// ---- POUs/VisMain/MAIN_VISION.TcPOU
PROGRAM MAIN_VISION
VAR
	fbPosCam1		: FB_PosImgSts;
	fbPosCam2		: FB_PosImgSts;
	fbPosCam3		: FB_PosImgSts;
	fbPosCam4		: FB_PosImgSts;
	fbPosCam5		: FB_PosImgSts;
	fbPosCam6		: FB_PosImgSts;
	fbPosCam7		: FB_PosImgSts;
	fbPosCam8		: FB_PosImgSts;
	fbPosCam9		: FB_PosImgSts;
	fbPosCam10		: FB_PosImgSts;
	
	fbMidStationCam	: FB_MidStaion;
	fbInfeedCam		: FB_InfeedCam;
	fbOutfeedCam	: FB_OutfeedCam;
	fbRejectCam		: FB_RejectCam;
	stPalletPosData	: ST_PalletImagingData;
	
	stMirrorDataSts1	: ST_Vis_Mirror;
	stMirrorDataSts2	: ST_Vis_Mirror;
	stMirrorDataSts3	: ST_Vis_Mirror;
	stMirrorDataSts4	: ST_Vis_Mirror;
	stMirrorDataSts5	: ST_Vis_Mirror;
	stMirrorDataSts6	: ST_Vis_Mirror;
	stMirrorDataSts7	: ST_Vis_Mirror;
	stMirrorDataSts8	: ST_Vis_Mirror;
	stMirrorDataSts9	: ST_Vis_Mirror;
	stMirrorDataSts10	: ST_Vis_Mirror;
	
	Cam1Trig : R_Trig;
	Cam2Trig : R_Trig;
	Cam3Trig : R_Trig;
	Cam4Trig : R_Trig; 
	Cam5Trig : R_Trig;
	Cam6Trig : R_Trig;
	Cam7Trig : R_Trig; 
	Cam8Trig : R_Trig;
	Cam9Trig : R_Trig; 
	Cam10Trig : R_Trig;
	CamMidStationTrig : R_Trig;
	CamInfeedTrig : R_Trig;
	CamOutfeedTrig : R_Trig;
	CamRejectTrig : R_Trig; 

	ImagingQueStep	: INT;
	
END_VAR


fbPosCam1(iStationId := 1 ,stPosData := stMirrorDataSts1, stAssemblyType := MAIN.stAssemblyData, nX := 830, nY := 980,stModuleHmi := MAIN.stModuleHmi );
fbPosCam2(iStationId := 2 ,stPosData := stMirrorDataSts2, stAssemblyType := MAIN.stAssemblyData, nX := 800, nY := 950,stModuleHmi := MAIN.stModuleHmi  );
fbPosCam3(iStationId := 3 ,stPosData := stMirrorDataSts3, stAssemblyType := MAIN.stAssemblyData, nX := 900, nY := 1010,stModuleHmi := MAIN.stModuleHmi  );
fbPosCam4(iStationId := 4 ,stPosData := stMirrorDataSts4, stAssemblyType := MAIN.stAssemblyData, nX := 890, nY := 950,stModuleHmi := MAIN.stModuleHmi  );
fbPosCam5(iStationId := 5 ,stPosData := stMirrorDataSts5, stAssemblyType := MAIN.stAssemblyData, nX := 840, nY := 1000,stModuleHmi := MAIN.stModuleHmi  );
fbPosCam6(iStationId := 6 ,stPosData := stMirrorDataSts6, stAssemblyType := MAIN.stAssemblyData, nX := 805, nY := 995,stModuleHmi := MAIN.stModuleHmi  );
fbPosCam7(iStationId := 7 ,stPosData := stMirrorDataSts7, stAssemblyType := MAIN.stAssemblyData, nX := 880, nY := 990,stModuleHmi := MAIN.stModuleHmi  );
fbPosCam8(iStationId := 8 ,stPosData := stMirrorDataSts8, stAssemblyType := MAIN.stAssemblyData, nX := 840, nY := 1010,stModuleHmi := MAIN.stModuleHmi  );
fbPosCam9(iStationId := 9 ,stPosData := stMirrorDataSts9, stAssemblyType := MAIN.stAssemblyData, nX := 850, nY := 990,stModuleHmi := MAIN.stModuleHmi  );
fbPosCam10(iStationId := 10 ,stPosData := stMirrorDataSts10, stAssemblyType := MAIN.stAssemblyData, nX := 860, nY := 1000,stModuleHmi := MAIN.stModuleHmi  );

fbMidStationCam(stRecipeData := MAIN.stAssemblyData, iStationId := MAIN.fbMeca500.iWorkingStation, stCouplerData := MAIN.stCouplerData);
fbInfeedCam(stPosData := stPalletPosData, stImagingSetValues := MAIN.stAssemblyData);
fbOutfeedCam();
fbRejectCam();

CASE ImagingQueStep OF
	0: ImagingQueStep := 1;// OFFLINE
	1: CamMidStationTrig(CLK := Trig.bMidStationCam);
		IF CamMidStationTrig.Q THEN
			fbMidStationCam.TrigImage();
		END_IF
		IF NOT Trig.bMidStationCam THEN
			ImagingQueStep := 2;
		END_IF
	2: CamInfeedTrig(CLK := Trig.bInfeedCam);
		IF CamInfeedTrig.Q THEN
			fbInfeedCam.TrigImage();
		END_IF
		IF NOT Trig.bInfeedCam THEN
			ImagingQueStep := 3;
		END_IF
	
	3:	CamOutfeedTrig(CLK := Trig.bOutfeedCam);
		IF CamOutfeedTrig.Q THEN
			fbOutfeedCam.TrigImage();
		END_IF
		IF NOT Trig.bOutfeedCam THEN
			ImagingQueStep := 4;
		END_IF
	
	4:	CamRejectTrig(CLK := Trig.bRejectCam);
		IF CamRejectTrig.Q THEN
			fbRejectCam.TrigImage();
		END_IF
		IF NOT Trig.bRejectCam THEN
			ImagingQueStep := 5;
		END_IF
	5: Cam1Trig(CLK := MAIN.stStation.fbSts1.bTrigPosCam);
		 IF Cam1Trig.Q THEN
			IF MAIN.stStation.fbSts1.bTrigPosCamLightTest THEN
				fbPosCam1.bTrigLightTestImage := TRUE;
			ELSIF MAIN.stStation.fbSts1.bTrigPosCamLaserTest THEN
				fbPosCam1.bTrigLaserTestImage := TRUE;
			ELSIF MAIN.stStation.fbSts1.bTrigPosCamCoupler THEN
				fbPosCam1.bTrigCouplerImage := TRUE;
			END_IF
			fbPosCam1.TrigImage();
		END_IF
		IF NOT MAIN.stStation.fbSts1.bTrigPosCam THEN
			stMirrorDataSts1.bDetectionFailed := FALSE;
			stMirrorDataSts1.bImagingDone := FALSE;
			ImagingQueStep := 6; 
		END_IF
		IF Cam1Trig.CLK THEN
			stMirrorDataSts1.bReadyForTrigger := FALSE;
		ELSE
			stMirrorDataSts1.bReadyForTrigger := TRUE;
		END_IF
		
	6:  Cam2Trig(CLK := MAIN.stStation.fbSts2.bTrigPosCam);
		IF Cam2Trig.Q THEN
			IF MAIN.stStation.fbSts2.bTrigPosCamLightTest THEN
				fbPosCam2.bTrigLightTestImage := TRUE;
			ELSIF MAIN.stStation.fbSts2.bTrigPosCamLaserTest THEN
				fbPosCam2.bTrigLaserTestImage := TRUE;
			ELSIF MAIN.stStation.fbSts2.bTrigPosCamCoupler THEN
				fbPosCam2.bTrigCouplerImage := TRUE;
			END_IF
			fbPosCam2.TrigImage();
		END_IF
	
		IF NOT MAIN.stStation.fbSts2.bTrigPosCam THEN
			stMirrorDataSts2.bDetectionFailed := FALSE;
			stMirrorDataSts2.bImagingDone := FALSE;
			ImagingQueStep := 7;
		END_IF
	
		IF Cam2Trig.CLK THEN
			stMirrorDataSts2.bReadyForTrigger := FALSE;
		ELSE
			stMirrorDataSts2.bReadyForTrigger := TRUE;
		END_IF
	
	
	7:  Cam3Trig(CLK := MAIN.stStation.fbSts3.bTrigPosCam);
		IF Cam3Trig.Q THEN
			IF MAIN.stStation.fbSts3.bTrigPosCamLightTest THEN
				fbPosCam3.bTrigLightTestImage := TRUE;
			ELSIF MAIN.stStation.fbSts3.bTrigPosCamLaserTest THEN
				fbPosCam3.bTrigLaserTestImage := TRUE;
			ELSIF MAIN.stStation.fbSts3.bTrigPosCamCoupler THEN
				fbPosCam3.bTrigCouplerImage := TRUE;
			END_IF
			fbPosCam3.TrigImage();
		END_IF
	
		IF NOT MAIN.stStation.fbSts3.bTrigPosCam THEN
			stMirrorDataSts3.bDetectionFailed := FALSE;
			stMirrorDataSts3.bImagingDone := FALSE;
			ImagingQueStep := 8;
		END_IF
	
		IF Cam3Trig.CLK THEN
			stMirrorDataSts3.bReadyForTrigger := FALSE;
		ELSE
			stMirrorDataSts3.bReadyForTrigger := TRUE;
		END_IF
	
	
	8:  Cam4Trig(CLK := MAIN.stStation.fbSts4.bTrigPosCam);
		IF Cam4Trig.Q THEN
			IF MAIN.stStation.fbSts4.bTrigPosCamLightTest THEN
				fbPosCam4.bTrigLightTestImage := TRUE;
			ELSIF MAIN.stStation.fbSts4.bTrigPosCamLaserTest THEN
				fbPosCam4.bTrigLaserTestImage := TRUE;
			ELSIF MAIN.stStation.fbSts4.bTrigPosCamCoupler THEN
				fbPosCam4.bTrigCouplerImage := TRUE;
			END_IF
			fbPosCam4.TrigImage();
		END_IF
	
		IF NOT MAIN.stStation.fbSts4.bTrigPosCam THEN
			stMirrorDataSts4.bDetectionFailed := FALSE;
			stMirrorDataSts4.bImagingDone := FALSE;
			ImagingQueStep := 9;
		END_IF
	
		IF Cam4Trig.CLK THEN
			stMirrorDataSts4.bReadyForTrigger := FALSE;
		ELSE
			stMirrorDataSts4.bReadyForTrigger := TRUE;
		END_IF
	
	
	9:  Cam5Trig(CLK := MAIN.stStation.fbSts5.bTrigPosCam);
		IF Cam5Trig.Q THEN
			IF MAIN.stStation.fbSts5.bTrigPosCamLightTest THEN
				fbPosCam5.bTrigLightTestImage := TRUE;
			ELSIF MAIN.stStation.fbSts5.bTrigPosCamLaserTest THEN
				fbPosCam5.bTrigLaserTestImage := TRUE;
			ELSIF MAIN.stStation.fbSts5.bTrigPosCamCoupler THEN
				fbPosCam5.bTrigCouplerImage := TRUE;
			END_IF
			fbPosCam5.TrigImage();
		END_IF
	
		IF NOT MAIN.stStation.fbSts5.bTrigPosCam THEN
			stMirrorDataSts5.bDetectionFailed := FALSE;
			stMirrorDataSts5.bImagingDone := FALSE;
			ImagingQueStep := 10;
		END_IF
	
		IF Cam5Trig.CLK THEN
			stMirrorDataSts5.bReadyForTrigger := FALSE;
		ELSE
			stMirrorDataSts5.bReadyForTrigger := TRUE;
		END_IF
	
	
	10: Cam6Trig(CLK := MAIN.stStation.fbSts6.bTrigPosCam);
		IF Cam6Trig.Q THEN
			IF MAIN.stStation.fbSts6.bTrigPosCamLightTest THEN
				fbPosCam6.bTrigLightTestImage := TRUE;
			ELSIF MAIN.stStation.fbSts6.bTrigPosCamLaserTest THEN
				fbPosCam6.bTrigLaserTestImage := TRUE;
			ELSIF MAIN.stStation.fbSts6.bTrigPosCamCoupler THEN
				fbPosCam6.bTrigCouplerImage := TRUE;
			END_IF
			fbPosCam6.TrigImage();
		END_IF
	
		IF NOT MAIN.stStation.fbSts6.bTrigPosCam THEN
			stMirrorDataSts6.bDetectionFailed := FALSE;
			stMirrorDataSts6.bImagingDone := FALSE;
			ImagingQueStep := 11;
		END_IF
	
		IF Cam6Trig.CLK THEN
			stMirrorDataSts6.bReadyForTrigger := FALSE;
		ELSE
			stMirrorDataSts6.bReadyForTrigger := TRUE;
		END_IF
	
	
	11: Cam7Trig(CLK := MAIN.stStation.fbSts7.bTrigPosCam);
		IF Cam7Trig.Q THEN
			IF MAIN.stStation.fbSts7.bTrigPosCamLightTest THEN
				fbPosCam7.bTrigLightTestImage := TRUE;
			ELSIF MAIN.stStation.fbSts7.bTrigPosCamLaserTest THEN
				fbPosCam7.bTrigLaserTestImage := TRUE;
			ELSIF MAIN.stStation.fbSts7.bTrigPosCamCoupler THEN
				fbPosCam7.bTrigCouplerImage := TRUE;
			END_IF
			fbPosCam7.TrigImage();
		END_IF
	
		IF NOT MAIN.stStation.fbSts7.bTrigPosCam THEN
			stMirrorDataSts7.bDetectionFailed := FALSE;
			stMirrorDataSts7.bImagingDone := FALSE;
			ImagingQueStep := 12;
		END_IF
	
		IF Cam7Trig.CLK THEN
			stMirrorDataSts7.bReadyForTrigger := FALSE;
		ELSE
			stMirrorDataSts7.bReadyForTrigger := TRUE;
		END_IF
	
	
	12: Cam8Trig(CLK := MAIN.stStation.fbSts8.bTrigPosCam);
		IF Cam8Trig.Q THEN
			IF MAIN.stStation.fbSts8.bTrigPosCamLightTest THEN
				fbPosCam8.bTrigLightTestImage := TRUE;
			ELSIF MAIN.stStation.fbSts8.bTrigPosCamLaserTest THEN
				fbPosCam8.bTrigLaserTestImage := TRUE;
			ELSIF MAIN.stStation.fbSts8.bTrigPosCamCoupler THEN
				fbPosCam8.bTrigCouplerImage := TRUE;
			END_IF
			fbPosCam8.TrigImage();
		END_IF
	
		IF NOT MAIN.stStation.fbSts8.bTrigPosCam THEN
			stMirrorDataSts8.bDetectionFailed := FALSE;
			stMirrorDataSts8.bImagingDone := FALSE;
			ImagingQueStep := 13;
		END_IF
	
		IF Cam8Trig.CLK THEN
			stMirrorDataSts8.bReadyForTrigger := FALSE;
		ELSE
			stMirrorDataSts8.bReadyForTrigger := TRUE;
		END_IF
	
	
	13: Cam9Trig(CLK := MAIN.stStation.fbSts9.bTrigPosCam);
		IF Cam9Trig.Q THEN
			IF MAIN.stStation.fbSts9.bTrigPosCamLightTest THEN
				fbPosCam9.bTrigLightTestImage := TRUE;
			ELSIF MAIN.stStation.fbSts9.bTrigPosCamLaserTest THEN
				fbPosCam9.bTrigLaserTestImage := TRUE;
			ELSIF MAIN.stStation.fbSts9.bTrigPosCamCoupler THEN
				fbPosCam9.bTrigCouplerImage := TRUE;
			END_IF
			fbPosCam9.TrigImage();
		END_IF
	
		IF NOT MAIN.stStation.fbSts9.bTrigPosCam THEN
			stMirrorDataSts9.bDetectionFailed := FALSE;
			stMirrorDataSts9.bImagingDone := FALSE;
			ImagingQueStep := 14;
		END_IF
	
		IF Cam9Trig.CLK THEN
			stMirrorDataSts9.bReadyForTrigger := FALSE;
		ELSE
			stMirrorDataSts9.bReadyForTrigger := TRUE;
		END_IF
	
	
	14: Cam10Trig(CLK := MAIN.stStation.fbSts10.bTrigPosCam);
		IF Cam10Trig.Q THEN
			IF MAIN.stStation.fbSts10.bTrigPosCamLightTest THEN
				fbPosCam10.bTrigLightTestImage := TRUE;
			ELSIF MAIN.stStation.fbSts10.bTrigPosCamLaserTest THEN
				fbPosCam10.bTrigLaserTestImage := TRUE;
			ELSIF MAIN.stStation.fbSts10.bTrigPosCamCoupler THEN
				fbPosCam10.bTrigCouplerImage := TRUE;
			END_IF
			fbPosCam10.TrigImage();
		END_IF
	
		IF NOT MAIN.stStation.fbSts10.bTrigPosCam THEN
			stMirrorDataSts10.bDetectionFailed := FALSE;
			stMirrorDataSts10.bImagingDone := FALSE;
			ImagingQueStep := 15;
		END_IF
	
		IF Cam10Trig.CLK THEN
			stMirrorDataSts10.bReadyForTrigger := FALSE;
		ELSE
			stMirrorDataSts10.bReadyForTrigger := TRUE;
		END_IF

	15: ImagingQueStep := 1;
	22: IF Trig.bInfeedCam THEN
			fbInfeedCam.TrigImage();
			Trig.bInfeedCam := FALSE;
		END_IF
END_CASE

END_PROGRAM

// ---- POUs/Sts/Vis/FB_PosImgSts.TcPOU
FUNCTION_BLOCK FB_PosImgSts
VAR_INPUT
	bTrigLightTestImage	: BOOL;
	bTrigLaserTestImage	: BOOL;
	bTrigCouplerImage		: BOOL;
	stPosData	: REFERENCE TO ST_Vis_Mirror;
	stAssemblyType : REFERENCE TO ST_Recipes;
	nX		: UDINT;
	nY		: UDINT;
	iStationId	: INT;
	stModuleHmi	: REFERENCE TO ST_ModuleHmi;
END_VAR
VAR_OUTPUT
	bImageReceived : BOOL;
	bPartDetectFailed : BOOL;
	iErrorId			: INT;
	bDone : BOOL;
END_VAR
VAR
	hr									: HRESULT;
	eVisionState						: ETcVnCameraState;
	fbCamera          					: FB_VN_GevCameraControl;
	ImageRawDisp						: ITcVnDisplayableImage;
	nNewImageCounter 					: UINT;
	ImageRaw							: Tc3_Vision.ITcVnImage;
	ipImageProsessed					: Tc3_Vision.ITcVnImage;
	ipImageProsessedDisp				: Tc3_Vision.ITcVnDisplayableImage;
	ipImageTest							: ITcVnImage;
	ipImageTestDisp						: ITcVnDisplayableImage;

	aStartPointCoupler1 				: TcVnPoint2_REAL;
	aEndPointCoupler1					: TcVnPoint2_REAL;
	
	ipEdgePointsCoupler1   				: ITcVnContainer;
	ipEdgePointsCoupler2				: ITcVnContainer;
	ipEdgePointsCoupler3				: ITcVnContainer;
	
	aStartPointCoupler2 				: TcVnPoint2_REAL;
	aEndPointCoupler2					: TcVnPoint2_REAL;
	aStartPointCoupler3 				: TcVnPoint2_REAL;
	aEndPointCoupler3					: TcVnPoint2_REAL;
	
	aStartPointMirror1 					: TcVnPoint2_REAL;
	aEndPointMirror1					: TcVnPoint2_REAL;
	aStartPointMirror2 					: TcVnPoint2_REAL;
	aEndPointMirror2					: TcVnPoint2_REAL;
	ipEdgePointsMirror1   				: ITcVnContainer;
	ipEdgePointsMirror2   				: ITcVnContainer;
	aElementMirror1						: TcVnPoint2_REAL;
	aElementMirror2						: TcVnPoint2_REAL;
	
	aMirrorEdgeCalc			: TcVnPoint2_REAL;
	aMirrorEdgeReal			: TcVnPoint2_REAL;
	

	
	rThreshold			: LREAL := 45;
	rMaxvalue			: LREAL := 255;

	stDetectionAreaLed						: TcVnRectangle_UDINT;
	stDetectionAreaLaser					: TcVnRectangle_UDINT;
	aAverageLed  							: TcVnVector4_LREAL;
	aAverageLaser  							: TcVnVector4_LREAL;
	aElementCoupler1 						: TcVnPoint2_REAL; 
	aElementCoupler2						: ARRAY [0..5] OF TcVnPoint2_REAL;
	aElementCoupler3						: ARRAY [0..5] OF TcVnPoint2_REAL;
	aCouplerAverage2						: TcVnPoint2_REAL;
	aCouplerAverage3						: TcVnPoint2_REAL;
	aCouplerCenterpoint						: TcVnPoint2_REAL;
	rWorldDistance							: LREAL;
	fbEventlogger							: FB_EventLogger;
	bInitTrig 								: BOOL;
	TrigCheckTmr							: TON;
END_VAR

fbEventlogger(stModuleHmi:=stModuleHmi);
eVisionState := fbCamera.GetState();

stDetectionAreaLed.nHeight := 200;
stDetectionAreaLed.nWidth := 200;
stDetectionAreaLed.nX := 1800;
stDetectionAreaLed.nY := 900;

stDetectionAreaLaser.nHeight := 20;
stDetectionAreaLaser.nWidth := 20;
stDetectionAreaLaser.nX := nX;
stDetectionAreaLaser.nY := nY;

bDone := FALSE;
bImageReceived := FALSE;
hr := 0;
TrigCheckTmr(PT := T#1S);


IF eVisionState = TCVN_CS_ERROR THEN
	hr := fbCamera.Reset();
ELSIF eVisionState = TCVN_CS_TRIGGERING THEN
	hr := fbCamera.TriggerImage();
ELSIF eVisionState < TCVN_CS_ACQUIRING THEN
    hr := fbCamera.StartAcquisition();
ELSIF eVisionState = TCVN_CS_ACQUIRING THEN
	hr := fbCamera.GetCurrentImageUndistorted(ImageRaw); 
	IF SUCCEEDED(hr) AND ImageRaw <> 0 THEN
		bPartDetectFailed := FALSE;
		bImageReceived := TRUE;
		nNewImageCounter := nNewImageCounter +1;
// 		hr := F_VN_CopyImage(ImageRaw, ipImageProsessed, hr);
// 		hr := F_VN_CopyIntoDisplayableImage (ImageRaw, ImageRawDisp, hr);
		bInitTrig := FALSE;
		TrigCheckTmr.IN := FALSE;
		hr := F_VN_ConvertColorSpace(ipSrcImage:= ImageRaw , ipDestImage:= ipImageProsessed ,
			eTransform:= ETcVnColorSpaceTransform.TCVN_CST_GRAY_TO_RGB, hrPrev:= hr);
		IF bTrigLightTestImage THEN
			hr := F_VN_CopyImage(ImageRaw, ipImageTest, hrPrev := hr);
			hr := F_VN_SetRoi_TcVnRectangle_UDINT(stRoi:= stDetectionAreaLed, ipDestImage:= ipImageTest, hrPrev:= hr);
			hr := F_VN_ImageAverage(ipSrcImage:= ipImageTest, aAverage:= aAverageLed, hrPrev:= hr);
			hr := F_VN_ResetRoi(ipImage:= ipImageTest, hrPrev:= hr);
			hr:= F_VN_ConvertColorSpace(ipSrcImage:= ipImageTest , ipDestImage:= ipImageTest ,
				eTransform:= ETcVnColorSpaceTransform.TCVN_CST_GRAY_TO_RGB, hrPrev:= hr);
			hr := F_VN_DrawRectangle_TcVnRectangle_UDINT(
				stRectangle:= stDetectionAreaLed,
				ipDestImage:= ipImageTest,
				aColor:= Color.Green,
				nThickness:= 1,
				hrPrev:= hr);
			hr := F_VN_CopyIntoDisplayableImage (ipImageTest, ipImageTestDisp, hr);	
			IF aAverageLed[0] > 230 THEN
				stPosData.bLightTestOk := TRUE;
				stPosData.bDetectionFailed := FALSE;
			ELSE
				stPosData.bLightTestOk := FALSE;
				stPosData.bDetectionFailed := TRUE;
			END_IF
			bTrigLightTestImage := FALSE;
		ELSIF bTrigLaserTestImage THEN
			hr := F_VN_CopyImage(ImageRaw, ipImageTest, hrPrev := hr);
			hr := F_VN_SetRoi_TcVnRectangle_UDINT(stRoi:= stDetectionAreaLaser, ipDestImage:= ipImageTest, hrPrev:= hr);
			hr := F_VN_ImageAverage(ipSrcImage:= ipImageTest, aAverage:= aAverageLaser, hrPrev:= hr);
			hr := F_VN_ResetRoi(ipImage:= ipImageTest, hrPrev:= hr);
			hr:= F_VN_ConvertColorSpace(ipSrcImage:= ipImageTest , ipDestImage:= ipImageTest ,
				eTransform:= ETcVnColorSpaceTransform.TCVN_CST_GRAY_TO_RGB, hrPrev:= hr);
			hr := F_VN_DrawRectangle_TcVnRectangle_UDINT(
				stRectangle:= stDetectionAreaLaser,
				ipDestImage:= ipImageTest,
				aColor:= Color.Green,
				nThickness:= 1,
				hrPrev:= hr);
			hr := F_VN_CopyIntoDisplayableImage (ipImageTest, ipImageTestDisp, hr);	
			IF aAverageLaser[0] > 230 THEN
				stPosData.bLaserTestOk := TRUE;
				stPosData.bDetectionFailed := FALSE;
			ELSE
				stPosData.bLaserTestOk := FALSE;
				stPosData.bDetectionFailed := TRUE;
			END_IF
			bTrigLaserTestImage := FALSE;
		ELSIF bTrigCouplerImage THEN	
			CouplerDetect();			
			bTrigCouplerImage := FALSE;
			stPosData.bImagingDone := TRUE;		
		ELSE
 			MirrorDetect();
			stPosData.bImagingDone := TRUE;	
		END_IF
	ELSIF bInitTrig AND TrigCheckTmr.Q THEN
		iErrorId := 304;
		fbEventlogger.bRaiseAlarm[11]:=TRUE;
		fbEventlogger.sErrorCode:= CONCAT(CONCAT('3', INT_TO_STRING(iStationId)), '4');
		bInitTrig := FALSE;
		TrigCheckTmr.IN := FALSE;
	END_IF
END_IF

METHOD CheckType : BOOL
VAR_INPUT
END_VAR
// CASE iStationId OF
// 	1..5: 
// 		IF stAssemblyType.Station1To5.sAssemblyType = 'AL-86068' THEN
// 			aStartPointCoupler1[0] := 750;
// 			aStartPointCoupler1[1] := 800;
// 			aEndPointCoupler1[0] := 750;
// 			aEndPointCoupler1[1] := 900;
// 			
// 			aStartPointCoupler2[0] := 750;
// 			aStartPointCoupler2[1] := 1170;
// 			aEndPointCoupler2[0] := 750;
// 			aEndPointCoupler2[1] := 1090;
// 		
// 			aStartPointMirror1[0] := 0;
// 			aStartPointMirror1[1] := 0;
// 			aEndPointMirror1[0] := 0;
// 			aEndPointMirror1[1] := 0;
// 			
// 			aStartPointMirror2[0] := 0;
// 			aStartPointMirror2[1] := 0;
// 			aEndPointMirror2[0] := 0;
// 			aEndPointMirror2[1] := 0;
// 		
// 		ELSIF stAssemblyType.Station1To5.sAssemblyType = 'AL-79710' THEN
// 			aStartPointCoupler1[0] := 770;
// 			aStartPointCoupler1[1] := 840;
// 			aEndPointCoupler1[0] := 770;
// 			aEndPointCoupler1[1] := 920;
// 			
// 			aStartPointCoupler2[0] := 770;
// 			aStartPointCoupler2[1] := 1150;
// 			aEndPointCoupler2[0] := 770;
// 			aEndPointCoupler2[1] := 1050;
// 		
// 			aStartPointMirror1[0] := 0;
// 			aStartPointMirror1[1] := 0;
// 			aEndPointMirror1[0] := 0;
// 			aEndPointMirror1[1] := 0;
// 			
// 			aStartPointMirror2[0] := 0;
// 			aStartPointMirror2[1] := 0;
// 			aEndPointMirror2[0] := 0;
// 			aEndPointMirror2[1] := 0;
// 		
// 		ELSIF stAssemblyType.Station1To5.sAssemblyType = 'AL-82028' THEN
// 			
// 			aStartPointCoupler1[0] := 750;
// 			aStartPointCoupler1[1] := 800;
// 			aEndPointCoupler1[0] := 750;
// 			aEndPointCoupler1[1] := 900;
// 			
// 			aStartPointCoupler2[0] := 750;
// 			aStartPointCoupler2[1] := 1170;
// 			aEndPointCoupler2[0] := 750;
// 			aEndPointCoupler2[1] := 1090;
// 		
// 			aStartPointMirror1[0] := 0;
// 			aStartPointMirror1[1] := 0;
// 			aEndPointMirror1[0] := 0;
// 			aEndPointMirror1[1] := 0;
// 			
// 			aStartPointMirror2[0] := 0;
// 			aStartPointMirror2[1] := 0;
// 			aEndPointMirror2[0] := 0;
// 			aEndPointMirror2[1] := 0;
// 		
// 		ELSIF stAssemblyType.Station1To5.sAssemblyType = 'AL-82026' THEN
// 			aStartPointCoupler[0] := ;
// 			aStartPointCoupler[1] := ;
// 			aEndPointCoupler[0] := ;
// 			aEndPointCoupler[1] := ;
// 		
// 			aStartPointMirror[0] := ;
// 			aStartPointMirror[1] := ;
// 			aEndPointMirror[0] := ;
// 			aEndPointMirror[1] := ;
// 		
// 		ELSIF stAssemblyType.Station1To5.sAssemblyType = 'AL-69219' THEN
// 			aStartPointCoupler1[0] := 793;
// 			aStartPointCoupler1[1] := 680;
// 			aEndPointCoupler1[0] := 793;
// 			aEndPointCoupler1[1] := 780;
// 			
// 			aStartPointCoupler2[0] := 793;
// 			aStartPointCoupler2[1] := 1330;
// 			aEndPointCoupler2[0] := 793;
// 			aEndPointCoupler2[1] := 1200;
// 		
// 			aStartPointMirror1[0] := 0;
// 			aStartPointMirror1[1] := 0;
// 			aEndPointMirror1[0] := 0;
// 			aEndPointMirror1[1] := 0;
// 			
// 			aStartPointMirror2[0] := 0;
// 			aStartPointMirror2[1] := 0;
// 			aEndPointMirror2[0] := 0;
// 			aEndPointMirror2[1] := 0;
// 		
// 		ELSIF stAssemblyType.Station1To5.sAssemblyType = 'AL-71449' THEN
// 			aStartPointCoupler[0] := ;
// 			aStartPointCoupler[1] := ;
// 			aEndPointCoupler[0] := ;
// 			aEndPointCoupler[1] := ;
// 		
// 			aStartPointMirror[0] := ;
// 			aStartPointMirror[1] := ;
// 			aEndPointMirror[0] := ;
// 			aEndPointMirror[1] := ;
// 		
// 		ELSIF stAssemblyType.Station1To5.sAssemblyType = 'AL-70918' THEN
// 			aStartPointCoupler[0] := ;
// 			aStartPointCoupler[1] := ;
// 			aEndPointCoupler[0] := ;
// 			aEndPointCoupler[1] := ;
// 		
// 			aStartPointMirror[0] := ;
// 			aStartPointMirror[1] := ;
// 			aEndPointMirror[0] := ;
// 			aEndPointMirror[1] := ;
// 		
// 		ELSIF stAssemblyType.Station1To5.sAssemblyType = 'AL-200617' THEN
// 			aStartPointCoupler1[0] := 770;
// 			aStartPointCoupler1[1] := 840;
// 			aEndPointCoupler1[0] := 770;
// 			aEndPointCoupler1[1] := 920;
// 			
// 			aStartPointCoupler2[0] := 770;
// 			aStartPointCoupler2[1] := 1150;
// 			aEndPointCoupler2[0] := 770;
// 			aEndPointCoupler2[1] := 1050;
// 		
// 			aStartPointMirror1[0] := 0;
// 			aStartPointMirror1[1] := 0;
// 			aEndPointMirror1[0] := 0;
// 			aEndPointMirror1[1] := 0;
// 			
// 			aStartPointMirror2[0] := 0;
// 			aStartPointMirror2[1] := 0;
// 			aEndPointMirror2[0] := 0;
// 			aEndPointMirror2[1] := 0;
// 		
// 		ELSIF stAssemblyType.Station1To5.sAssemblyType = 'AL-200613' THEN
// 			aStartPointCoupler1[0] := 793;
// 			aStartPointCoupler1[1] := 680;
// 			aEndPointCoupler1[0] := 793;
// 			aEndPointCoupler1[1] := 780;
// 			
// 			aStartPointCoupler2[0] := 793;
// 			aStartPointCoupler2[1] := 1330;
// 			aEndPointCoupler2[0] := 793;
// 			aEndPointCoupler2[1] := 1200;
// 		
// 			aStartPointMirror1[0] := 0;
// 			aStartPointMirror1[1] := 0;
// 			aEndPointMirror1[0] := 0;
// 			aEndPointMirror1[1] := 0;
// 			
// 			aStartPointMirror2[0] := 0;
// 			aStartPointMirror2[1] := 0;
// 			aEndPointMirror2[0] := 0;
// 			aEndPointMirror2[1] := 0;
// 		
// 		ELSIF stAssemblyType.Station1To5.sAssemblyType = 'AL-88450' THEN
// 			aStartPointCoupler[0] := ;
// 			aStartPointCoupler[1] := ;
// 			aEndPointCoupler[0] := ;
// 			aEndPointCoupler[1] := ;
// 		
// 			aStartPointMirror[0] := ;
// 			aStartPointMirror[1] := ;
// 			aEndPointMirror[0] := ;
// 			aEndPointMirror[1] := ;
// 		
// 		ELSIF stAssemblyType.Station1To5.sAssemblyType = 'AL-200665' THEN
// 			aStartPointCoupler1[0] := 644;
// 			aStartPointCoupler1[1] := 780;
// 			aEndPointCoupler1[0] := 644;
// 			aEndPointCoupler1[1] := 780;
// 			
// 			aStartPointCoupler2[0] := 644;
// 			aStartPointCoupler2[1] := 1210;
// 			aEndPointCoupler2[0] := 644;
// 			aEndPointCoupler2[1] := 1100;
// 		
// 			aStartPointMirror1[0] := 0;
// 			aStartPointMirror1[1] := 0;
// 			aEndPointMirror1[0] := 0;
// 			aEndPointMirror1[1] := 0;
// 			
// 			aStartPointMirror2[0] := 0;
// 			aStartPointMirror2[1] := 0;
// 			aEndPointMirror2[0] := 0;
// 			aEndPointMirror2[1] := 0;
// 		
// 		ELSIF stAssemblyType.Station1To5.sAssemblyType = 'AL-200663' THEN
// 			aStartPointCoupler1[0] := 644;
// 			aStartPointCoupler1[1] := 780;
// 			aEndPointCoupler1[0] := 644;
// 			aEndPointCoupler1[1] := 780;
// 			
// 			aStartPointCoupler2[0] := 644;
// 			aStartPointCoupler2[1] := 1210;
// 			aEndPointCoupler2[0] := 644;
// 			aEndPointCoupler2[1] := 1100;
// 		
// 			aStartPointMirror1[0] := 0;
// 			aStartPointMirror1[1] := 0;
// 			aEndPointMirror1[0] := 0;
// 			aEndPointMirror1[1] := 0;
// 			
// 			aStartPointMirror2[0] := 0;
// 			aStartPointMirror2[1] := 0;
// 			aEndPointMirror2[0] := 0;
// 			aEndPointMirror2[1] := 0;
// 		
// 		ELSIF stAssemblyType.Station1To5.sAssemblyType = 'AL-82029' THEN
// 			aStartPointCoupler1[0] := 750;
// 			aStartPointCoupler1[1] := 800;
// 			aEndPointCoupler1[0] := 750;
// 			aEndPointCoupler1[1] := 900;
// 			
// 			aStartPointCoupler2[0] := 750;
// 			aStartPointCoupler2[1] := 1170;
// 			aEndPointCoupler2[0] := 750;
// 			aEndPointCoupler2[1] := 1090;
// 		
// 			aStartPointMirror1[0] := 0;
// 			aStartPointMirror1[1] := 0;
// 			aEndPointMirror1[0] := 0;
// 			aEndPointMirror1[1] := 0;
// 			
// 			aStartPointMirror2[0] := 0;
// 			aStartPointMirror2[1] := 0;
// 			aEndPointMirror2[0] := 0;
// 			aEndPointMirror2[1] := 0;
// 		
// 		ELSIF stAssemblyType.Station1To5.sAssemblyType = 'AL-86069' THEN
// 			aStartPointCoupler1[0] := 750;
// 			aStartPointCoupler1[1] := 800;
// 			aEndPointCoupler1[0] := 750;
// 			aEndPointCoupler1[1] := 900;
// 			
// 			aStartPointCoupler2[0] := 750;
// 			aStartPointCoupler2[1] := 1170;
// 			aEndPointCoupler2[0] := 750;
// 			aEndPointCoupler2[1] := 1090;
// 		
// 			aStartPointMirror1[0] := 0;
// 			aStartPointMirror1[1] := 0;
// 			aEndPointMirror1[0] := 0;
// 			aEndPointMirror1[1] := 0;
// 			
// 			aStartPointMirror2[0] := 0;
// 			aStartPointMirror2[1] := 0;
// 			aEndPointMirror2[0] := 0;
// 			aEndPointMirror2[1] := 0;
// 		
// 		ELSIF stAssemblyType.Station1To5.sAssemblyType = 'AL-79420' THEN
// 			aStartPointCoupler1[0] := 770;
// 			aStartPointCoupler1[1] := 840;
// 			aEndPointCoupler1[0] := 770;
// 			aEndPointCoupler1[1] := 920;
// 			
// 			aStartPointCoupler2[0] := 770;
// 			aStartPointCoupler2[1] := 1150;
// 			aEndPointCoupler2[0] := 770;
// 			aEndPointCoupler2[1] := 1050;
// 		
// 			aStartPointMirror1[0] := 0;
// 			aStartPointMirror1[1] := 0;
// 			aEndPointMirror1[0] := 0;
// 			aEndPointMirror1[1] := 0;
// 			
// 			aStartPointMirror2[0] := 0;
// 			aStartPointMirror2[1] := 0;
// 			aEndPointMirror2[0] := 0;
// 			aEndPointMirror2[1] := 0;
// 		
// 		ELSIF stAssemblyType.Station1To5.sAssemblyType = 'AL-82027' THEN
// 			aStartPointCoupler[0] := ;
// 			aStartPointCoupler[1] := ;
// 			aEndPointCoupler[0] := ;
// 			aEndPointCoupler[1] := ;
// 		
// 			aStartPointMirror[0] := ;
// 			aStartPointMirror[1] := ;
// 			aEndPointMirror[0] := ;
// 			aEndPointMirror[1] := ;
// 		
// 		ELSIF stAssemblyType.Station1To5.sAssemblyType = 'AL-69220' THEN
// 			aStartPointCoupler1[0] := 793;
// 			aStartPointCoupler1[1] := 680;
// 			aEndPointCoupler1[0] := 793;
// 			aEndPointCoupler1[1] := 780;
// 			
// 			aStartPointCoupler2[0] := 793;
// 			aStartPointCoupler2[1] := 1330;
// 			aEndPointCoupler2[0] := 793;
// 			aEndPointCoupler2[1] := 1200;
// 		
// 			aStartPointMirror1[0] := 0;
// 			aStartPointMirror1[1] := 0;
// 			aEndPointMirror1[0] := 0;
// 			aEndPointMirror1[1] := 0;
// 			
// 			aStartPointMirror2[0] := 0;
// 			aStartPointMirror2[1] := 0;
// 			aEndPointMirror2[0] := 0;
// 			aEndPointMirror2[1] := 0;
// 		
// 		ELSIF stAssemblyType.Station1To5.sAssemblyType = 'AL-71450' THEN
// 			aStartPointCoupler[0] := ;
// 			aStartPointCoupler[1] := ;
// 			aEndPointCoupler[0] := ;
// 			aEndPointCoupler[1] := ;
// 		
// 			aStartPointMirror[0] := ;
// 			aStartPointMirror[1] := ;
// 			aEndPointMirror[0] := ;
// 			aEndPointMirror[1] := ;
// 		
// 		ELSIF stAssemblyType.Station1To5.sAssemblyType = 'AL-70916' THEN
// 			aStartPointCoupler[0] := ;
// 			aStartPointCoupler[1] := ;
// 			aEndPointCoupler[0] := ;
// 			aEndPointCoupler[1] := ;
// 		
// 			aStartPointMirror[0] := ;
// 			aStartPointMirror[1] := ;
// 			aEndPointMirror[0] := ;
// 			aEndPointMirror[1] := ;
// 		
// 		ELSIF stAssemblyType.Station1To5.sAssemblyType = 'AL-200618' THEN
// 			aStartPointCoupler1[0] := 770;
// 			aStartPointCoupler1[1] := 840;
// 			aEndPointCoupler1[0] := 770;
// 			aEndPointCoupler1[1] := 920;
// 			
// 			aStartPointCoupler2[0] := 770;
// 			aStartPointCoupler2[1] := 1150;
// 			aEndPointCoupler2[0] := 770;
// 			aEndPointCoupler2[1] := 1050;
// 		
// 			aStartPointMirror1[0] := 0;
// 			aStartPointMirror1[1] := 0;
// 			aEndPointMirror1[0] := 0;
// 			aEndPointMirror1[1] := 0;
// 			
// 			aStartPointMirror2[0] := 0;
// 			aStartPointMirror2[1] := 0;
// 			aEndPointMirror2[0] := 0;
// 			aEndPointMirror2[1] := 0;
// 		
// 		ELSIF stAssemblyType.Station1To5.sAssemblyType = 'AL-200614' THEN
// 			aStartPointCoupler1[0] := 793;
// 			aStartPointCoupler1[1] := 680;
// 			aEndPointCoupler1[0] := 793;
// 			aEndPointCoupler1[1] := 780;
// 			
// 			aStartPointCoupler2[0] := 793;
// 			aStartPointCoupler2[1] := 1330;
// 			aEndPointCoupler2[0] := 793;
// 			aEndPointCoupler2[1] := 1200;
// 		
// 			aStartPointMirror1[0] := 0;
// 			aStartPointMirror1[1] := 0;
// 			aEndPointMirror1[0] := 0;
// 			aEndPointMirror1[1] := 0;
// 			
// 			aStartPointMirror2[0] := 0;
// 			aStartPointMirror2[1] := 0;
// 			aEndPointMirror2[0] := 0;
// 			aEndPointMirror2[1] := 0;
// 		
// 		ELSIF stAssemblyType.Station1To5.sAssemblyType = 'AL-88470' THEN
// 			aStartPointCoupler[0] := ;
// 			aStartPointCoupler[1] := ;
// 			aEndPointCoupler[0] := ;
// 			aEndPointCoupler[1] := ;
// 		
// 			aStartPointMirror[0] := ;
// 			aStartPointMirror[1] := ;
// 			aEndPointMirror[0] := ;
// 			aEndPointMirror[1] := ;
// 		
// 		ELSIF stAssemblyType.Station1To5.sAssemblyType = 'AL-200662' THEN
// 			aStartPointCoupler1[0] := 644;
// 			aStartPointCoupler1[1] := 780;
// 			aEndPointCoupler1[0] := 644;
// 			aEndPointCoupler1[1] := 780;
// 			
// 			aStartPointCoupler2[0] := 644;
// 			aStartPointCoupler2[1] := 1210;
// 			aEndPointCoupler2[0] := 644;
// 			aEndPointCoupler2[1] := 1100;
// 		
// 			aStartPointMirror1[0] := 0;
// 			aStartPointMirror1[1] := 0;
// 			aEndPointMirror1[0] := 0;
// 			aEndPointMirror1[1] := 0;
// 			
// 			aStartPointMirror2[0] := 0;
// 			aStartPointMirror2[1] := 0;
// 			aEndPointMirror2[0] := 0;
// 			aEndPointMirror2[1] := 0;
// 		
// 		ELSIF stAssemblyType.Station1To5.sAssemblyType = 'AL-200664' THEN
// 			aStartPointCoupler1[0] := 644;
// 			aStartPointCoupler1[1] := 780;
// 			aEndPointCoupler1[0] := 644;
// 			aEndPointCoupler1[1] := 780;
// 			
// 			aStartPointCoupler2[0] := 644;
// 			aStartPointCoupler2[1] := 1210;
// 			aEndPointCoupler2[0] := 644;
// 			aEndPointCoupler2[1] := 1100;
// 		
// 			aStartPointMirror1[0] := 0;
// 			aStartPointMirror1[1] := 0;
// 			aEndPointMirror1[0] := 0;
// 			aEndPointMirror1[1] := 0;
// 			
// 			aStartPointMirror2[0] := 0;
// 			aStartPointMirror2[1] := 0;
// 			aEndPointMirror2[0] := 0;
// 			aEndPointMirror2[1] := 0;
// 		
// 		END_IF;
// 
// END_CASE
END_METHOD

METHOD CouplerDetect : BOOL

VAR
	bCheckOnce 					: BOOL := TRUE;
	hrEdgeT						: HRESULT;
	nIndex						: ULINT;
	
END_VAR
hrEdgeT := 0;

aStartPointCoupler1[0] := 1000;
aStartPointCoupler1[1] := 1000;
aEndPointCoupler1[0] := 550;
aEndPointCoupler1[1] := 1000;

		
hrEdgeT := F_VN_LocateEdge(
	ipSrcImage:= ImageRaw, 
	ipEdgePoints:= ipEdgePointsCoupler1, 
	aStartPoint:= aStartPointCoupler1, 
	aEndPoint:= aEndPointCoupler1, 
	eEdgeDirection:= ETcVnEdgeDirection.TCVN_ED_Light_TO_Dark, 
	fMinStrength:= 45, 
	nSearchLines:= 5, 
	hrPrev:= hr, 
	fAvgStrength=> );
	
hrEdgeT := F_VN_GetAt_TcVnVector2_REAL(ipContainer:= ipEdgePointsCoupler1, aElement:= aElementCoupler1, nIndex:= 0, hrPrev:= hrEdgeT);
	
aStartPointCoupler2[0] := aElementCoupler1[0]-40;
aStartPointCoupler2[1] := 600;
aEndPointCoupler2[0] := aElementCoupler1[0]-40;
aEndPointCoupler2[1] := 1000;	

aStartPointCoupler3[0] := aElementCoupler1[0]-40;
aStartPointCoupler3[1] := 1400;
aEndPointCoupler3[0] := aElementCoupler1[0]-40;
aEndPointCoupler3[1] := 1000;	

hrEdgeT := F_VN_LocateEdge(
	ipSrcImage:= ImageRaw, 
	ipEdgePoints:= ipEdgePointsCoupler2, 
	aStartPoint:= aStartPointCoupler2, 
	aEndPoint:= aEndPointCoupler2, 
	eEdgeDirection:= ETcVnEdgeDirection.TCVN_ED_Light_TO_Dark, 
	fMinStrength:= 45, 
	nSearchLines:= 4, 
	hrPrev:= hr, 
	fAvgStrength=> );
hrEdgeT := F_VN_LocateEdge(
	ipSrcImage:= ImageRaw, 
	ipEdgePoints:= ipEdgePointsCoupler3, 
	aStartPoint:= aStartPointCoupler3, 
	aEndPoint:= aEndPointCoupler3, 
	eEdgeDirection:= ETcVnEdgeDirection.TCVN_ED_Light_TO_Dark, 
	fMinStrength:= 45, 
	nSearchLines:= 4, 
	hrPrev:= hr, 
	fAvgStrength=> );
IF SUCCEEDED(hrEdgeT) THEN
	hrEdgeT := F_VN_DrawPoints(
		ipPoints:= ipEdgePointsCoupler1, 
		ipDestImage:= ipImageProsessed, 
		eShape:= ETcVnDrawShape.TCVN_DS_X, 
		aColor:= Color.Lime, 
		hrPrev:= hr);

	hrEdgeT := F_VN_DrawPoints(
		ipPoints:= ipEdgePointsCoupler2, 
		ipDestImage:= ipImageProsessed, 
		eShape:= ETcVnDrawShape.TCVN_DS_X, 
		aColor:= Color.Lime, 
		hrPrev:= hr);
		
	hrEdgeT := F_VN_DrawPoints(
		ipPoints:= ipEdgePointsCoupler3, 
		ipDestImage:= ipImageProsessed, 
		eShape:= ETcVnDrawShape.TCVN_DS_X, 
		aColor:= Color.Lime, 
		hrPrev:= hr);
	FOR nIndex := 0 TO 4 DO
		hrEdgeT := F_VN_GetAt_TcVnVector2_REAL(ipContainer:= ipEdgePointsCoupler2, aElement:= aElementCoupler2[nIndex], nIndex:= nIndex, hrPrev:= hrEdgeT);
		hrEdgeT := F_VN_GetAt_TcVnVector2_REAL(ipContainer:= ipEdgePointsCoupler3, aElement:= aElementCoupler3[nIndex], nIndex:= nIndex, hrPrev:= hrEdgeT);
	END_FOR
	aCouplerAverage2[0] := REAL_TO_ULINT((aElementCoupler2[0][0] + aElementCoupler2[1][0] + aElementCoupler2[2][0] + aElementCoupler2[3][0]+ aElementCoupler2[4][0] )/ 5);
	aCouplerAverage2[1] := REAL_TO_ULINT((aElementCoupler2[0][1] + aElementCoupler2[1][1] + aElementCoupler2[2][1] + aElementCoupler2[3][1]+ aElementCoupler2[4][1] )/ 5);
	aCouplerAverage3[0] := REAL_TO_ULINT((aElementCoupler3[0][0] + aElementCoupler3[1][0] + aElementCoupler3[2][0] + aElementCoupler3[3][0]+ aElementCoupler3[4][0] )/ 5);
	aCouplerAverage3[1] := REAL_TO_ULINT((aElementCoupler3[0][1] + aElementCoupler3[1][1] + aElementCoupler3[2][1] + aElementCoupler3[3][1]+ aElementCoupler3[4][1] )/ 5);
	aCouplerCenterpoint[0] := (aCouplerAverage2[0] + aCouplerAverage3[0])/2;
	aCouplerCenterpoint[1] := (aCouplerAverage2[1] + aCouplerAverage3[1])/2;
	hr := F_VN_CopyIntoDisplayableImage (ipImageProsessed, ipImageProsessedDisp, hr);
	
	
ELSE
	IF bCheckOnce THEN
		ADSLOGSTR(msgCtrlMask := ADSLOG_MSGTYPE_ERROR, msgFmtStr := 'Error1', strArg:= ' ');
		bCheckOnce := FALSE;
	END_IF
END_IF
END_METHOD

METHOD MirrorDetect : BOOL
VAR_INPUT
END_VAR
VAR
	aPoint1 : TcVnPoint2_REAL := [0,0];
	aPoint2 : TcVnPoint2_REAL := [0,1];	
	
  	aCameraMatrix           : TcVnMatrix3x3_LREAL;
    aDistortionCoefficients : TcVnArray8_LREAL;
    aRotationMatrix         : TcVnMatrix3x3_LREAL;
    aTranslationVector      : TcVnVector3_LREAL;
	

END_VAR
fbCamera.GetCameraMatrix(aCameraMatrix := aCameraMatrix);
fbCamera.GetDistortionCoefficients(aDistortionCoefficients := aDistortionCoefficients);
fbCamera.GetRotationMatrix(aRotationMatrix := aRotationMatrix);
fbCamera.GetTranslationVector(aTranslationVector := aTranslationVector);

hr := F_VN_ImagePointsWorldDistance( 
	aImagePoint1 := aPoint1,
	aImagePoint2 := aPoint2,
	fWorldDistance := rWorldDistance,
	aCameraMatrix := aCameraMatrix,
	aDistortionCoefficients := aDistortionCoefficients,
	aRotationMatrix := aRotationMatrix,
	aTranslationVector := aTranslationVector,
	fZ := 0,
	hrPrev := hr);
	

CASE iStationId OF
 	1..5:
	aMirrorEdgeCalc[1] := stAssemblyType.Station1To5.rMirrorCenterOffsetToWeightCenterY/rWorldDistance; // calculates the distance in px of the mirror centerpoint to weight centerpoint. Is used to determine currect positioning of the mirror 
	
	// Detection from center to upper edge
	aStartPointMirror1[0] := aCouplerCenterpoint[0] - ((stAssemblyType.Station1To5.rCouplerGroveDepth)/rWorldDistance) + (stAssemblyType.Station1To5.rMirrorGripPointOffsetToEdgeX/rWorldDistance) ;
	aStartPointMirror1[1] := aCouplerCenterpoint[1]; // Coupler centerpoint based Y Startpoint
	aEndPointMirror1[0] := aStartPointMirror1[0];
	aEndPointMirror1[1] := aCouplerCenterpoint[1] - (((stAssemblyType.Station1To5.rMirrorDimensions[1]/2) - stAssemblyType.Station1To5.rMirrorCenterOffsetToWeightCenterY)/rWorldDistance)-100; // endpoint based on coupler centerpoint - mirror weight centerpoint to edge width + some extra
	// detection from center to lower edge
	aStartPointMirror2[0] := aCouplerCenterpoint[0] - ((stAssemblyType.Station1To5.rCouplerGroveDepth)/rWorldDistance) + (stAssemblyType.Station1To5.rMirrorGripPointOffsetToEdgeX/rWorldDistance);
	aStartPointMirror2[1] := aCouplerCenterpoint[1];
	aEndPointMirror2[0] := aStartPointMirror2[0];
	aEndPointMirror2[1] := aCouplerCenterpoint[1] + (((stAssemblyType.Station1To5.rMirrorDimensions[1]/2) - stAssemblyType.Station1To5.rMirrorCenterOffsetToWeightCenterY)/rWorldDistance)+100;
	
	6..10:
	aStartPointMirror1[0] := 0;
	aStartPointMirror1[1] := 0;
	aEndPointMirror1[0] := 0;
	aEndPointMirror1[1] := 0;
			
	aStartPointMirror2[0] := 0;
	aStartPointMirror2[1] := 0;
	aEndPointMirror2[0] := 0;
	aEndPointMirror2[1] := 0;
END_CASE

hr := F_VN_LocateEdge(
	ipSrcImage:= ImageRaw, 
	ipEdgePoints:= ipEdgePointsMirror1, 
	aStartPoint:= aStartPointMirror1, 
	aEndPoint:= aEndPointMirror1, 
	eEdgeDirection:= ETcVnEdgeDirection.TCVN_ED_DARK_TO_LIGHT, 
	fMinStrength:= 45, 
	nSearchLines:= 1, 
	hrPrev:= hr, 
	fAvgStrength=> );
hr := F_VN_LocateEdge(
	ipSrcImage:= ImageRaw, 
	ipEdgePoints:= ipEdgePointsMirror2, 
	aStartPoint:= aStartPointMirror2, 
	aEndPoint:= aEndPointMirror2, 
	eEdgeDirection:= ETcVnEdgeDirection.TCVN_ED_DARK_TO_LIGHT, 
	fMinStrength:= 45, 
	nSearchLines:= 1, 
	hrPrev:= hr, 
	fAvgStrength=> );
	IF SUCCEEDED(hr) THEN
		hr := F_VN_GetAt_TcVnVector2_REAL(ipContainer:= ipEdgePointsMirror1, aElement:= aElementMirror1, nIndex:= 0, hrPrev:= hr);
		hr := F_VN_GetAt_TcVnVector2_REAL(ipContainer:= ipEdgePointsMirror2, aElement:= aElementMirror2, nIndex:= 0, hrPrev:= hr);
		hr := F_VN_DrawPoints(
			ipPoints:= ipEdgePointsMirror1, 
			ipDestImage:= ipImageProsessed, 
			eShape:= ETcVnDrawShape.TCVN_DS_X, 
			aColor:= Color.Lime, 
			hrPrev:= hr);
		hr := F_VN_DrawPoints(
			ipPoints:= ipEdgePointsMirror2, 
			ipDestImage:= ipImageProsessed, 
			eShape:= ETcVnDrawShape.TCVN_DS_X, 
			aColor:= Color.Lime, 
			hrPrev:= hr);
		stPosData.rMirrorOffsetToCalPoints[1] := (( aCouplerCenterpoint[1]) - ((aElementMirror1[1] + aElementMirror2[1])/2) - aMirrorEdgeCalc[1])*rWorldDistance;
		hr := F_VN_CopyIntoDisplayableImage (ipImageProsessed, ipImageProsessedDisp, hr);
	END_IF
END_METHOD

METHOD TrigImage : BOOL
VAR_INPUT
END_VAR
fbCamera.TriggerImage();
bInitTrig := TRUE;
TrigCheckTmr.IN := TRUE;
END_METHOD

END_FUNCTION_BLOCK

// ---- POUs/VisMain/FB_MidStaion.TcPOU
FUNCTION_BLOCK FB_MidStaion
VAR_INPUT
	bTriggerImage : BOOL;
 	stRecipeData: REFERENCE TO ST_Recipes;
	stCouplerData		: REFERENCE TO ST_CouplerImagingData;
	iStationId			: INT;
END_VAR
VAR_OUTPUT
	bError : BOOL;
END_VAR
VAR
	hr									: HRESULT;
	eVisionState						: ETcVnCameraState;
	fbCamera          					: FB_VN_GevCameraControl;
	ImageRawDisp						: ITcVnDisplayableImage;
	ImageFilter							: Tc3_Vision.ITcVnImage;
	ImageFilterDisp						: ITcVnDisplayableImage;
	nNewImageCounter 					: UINT;
	ImageRaw: Tc3_Vision.ITcVnImage;
	ipImageProsessed					: Tc3_Vision.ITcVnImage;
	
	nFilterWidth						: UDINT := 7;
	fTargetRadius						: REAL := 250;		// Hakuympyrän oletettu säde (=moottorin säde), tämä reseptiin
	fMinRadius							: REAL := 150;		// Hakuympyrän pienin sallittu säde, tämä reseptiin
	

	aElement1 							: TcVnPoint2_REAL;
	aElement2							: TcVnPoint2_REAL;
	ipEdgePointsL    					: ITcVnContainer;
	ipEdgePointsR    					: ITcVnContainer;
	eAlgorithm           				: ETcVnEdgeDetectionAlgorithm;
	aFitlineL							: TcVnVector4_LREAL;
	aFitlineR							: TcVnVector4_LREAL;
	
	aStartPointCoupler					: TcVnPoint2_REAL;
	aEndPointCoupler					: TcVnPoint2_REAL;
	aStartPoint1 						: TcVnPoint2_REAL;
	aEndPoint1							: TcVnPoint2_REAL;
	aStartPoint2 						: TcVnPoint2_REAL;
	aEndPoint2							: TcVnPoint2_REAL;
	aStartPoint3 						: TcVnPoint2_REAL;
	aEndPoint3							: TcVnPoint2_REAL;
	rClawLLineAngleRad						: LREAL;
	rClawLLineAngleDeg						: LREAL;
	rClawRLineAngleRad						: LREAL;
	rClawRLineAngleDeg						: LREAL;
	rSearchLineDist							: REAL := 10;
	
	rLineAngleRad						: LREAL;
	rLineAngleDeg						: LREAL;
	rLineAngleResultDeg					: LREAL;
	aCenter								: TcVnPoint2_REAL;
	ipContourPoints						: ITcVnContainer;
	stMotorEllipse						: TcVnRotatedRectangle;
	ipImageProsessedDisp				: Tc3_Vision.ITcVnDisplayableImage;
	
	bGreatSuccess: BOOL;
	bSuccess_ImageTransform: BOOL;
	bSuccess_LeftLocate: BOOL;
	bSuccess_RightLocate: BOOL;
	bSuccess_DrawCircle: BOOL;
	bSuccess_FindEllipse: BOOL;
	bSuccess_FixtureMethod : BOOL;
	
	

	
	rThreshold			: LREAL := 45;
	rMaxvalue			: LREAL := 255;
	
	
	// RMSE
	slope     : LREAL;  // a
    intercept : LREAL;  // b
    rmsError  : LREAL;  
	bRmsErr : BOOL;
	
END_VAR

VAR RETAIN
	bModeFixtureToGripper: BOOL := TRUE;
END_VAR

eVisionState := fbCamera.GetState();


stCouplerData.bImageReceived := FALSE;
hr := 0;



IF eVisionState = TCVN_CS_ERROR THEN
	hr := fbCamera.Reset();
ELSIF eVisionState = TCVN_CS_TRIGGERING THEN
	hr := fbCamera.TriggerImage();
ELSIF eVisionState < TCVN_CS_ACQUIRING THEN
    hr := fbCamera.StartAcquisition();
ELSIF eVisionState = TCVN_CS_ACQUIRING THEN
	hr := fbCamera.GetCurrentImage(ImageRaw); // switch to undistorted
	IF SUCCEEDED(hr) AND ImageRaw <> 0 THEN
		bError := FALSE;
		stCouplerData.bImagingDone := FALSE;
		stCouplerData.bPartDetectFailed := FALSE;
		stCouplerData.bPartDetectSucceeded := FALSE;
		stCouplerData.bImageReceived := TRUE;
		SetParams();
		nNewImageCounter := nNewImageCounter +1;
		//hr := F_VN_CopyIntoDisplayableImage (ImageRaw, ImageRawDisp, hr);
		bSuccess_FixtureMethod := FALSE;
		FixtureGripper();
		bSuccess_FixtureMethod := SUCCEEDED(hr);
		IF NOT bSuccess_FixtureMethod THEN
			Err.Err; // PALLET IMAGING ERROR
		ELSE
			hr := F_VN_CopyIntoDisplayableImage (ipImageProsessed, ipImageProsessedDisp, hr);	
			stCouplerData.bImagingDone := TRUE;
		END_IF
 		hr := F_VN_CopyIntoDisplayableImage (ImageRaw, ImageRawDisp, hr);
// 		hr := F_VN_CopyIntoDisplayableImage (ImageFilter, ImageFilterDisp, hr);

	ELSE
		bError := TRUE;
		Err.Err; // PALLET IMAGING ERROR
	END_IF
END_IF

METHOD FixtureGripper : BOOL
VAR_INPUT

END_VAR

VAR
	fFoundStr : REAL;
	x : ARRAY[1..10] OF LREAL;
    y : ARRAY[1..10] OF LREAL;
	i : UDINT;
END_VAR

//
//	PARAMETERS
//

// left claw search area, Search dir right-to-left
aEndPoint1[0] 	:= 800;
aEndPoint1[1] 	:= 600;
aStartPoint1[0] := 1100;
aStartPoint1[1] := 600;

// Right claw search area, Search dir left-to-right
aStartPoint2[0] := 1080;
aStartPoint2[1] := 600;
aEndPoint2[0] 	:= 1400;
aEndPoint2[1] 	:= 600;

// Claw bottom search area, search dir bottom up
aStartPoint3[0] := 1150;
aStartPoint3[1] := 600;
aEndPoint3[0] 	:= 1400;
aEndPoint3[1] 	:= 600;

// Motor Circle finding
aCenter[0]		:= 1110;
aCenter[1]		:= 1125;

// Coupler edge find, in relation to found motor center
// aStartPointCoupler[0] 	:= 0; // 100
// aStartPointCoupler[1] 	:= 120; //-150
// aEndPointCoupler[0]		:= 0;
// aEndPointCoupler[1]		:= 0; // -70

//  //Start values FOR 69636
// aStartPointCoupler[0] 	:= 0;
// aStartPointCoupler[1] 	:= 90;
// aEndPointCoupler[0]		:= 0;
// aEndPointCoupler[1]		:= 250;

//  //Start values FOR AL-78676
// aStartPointCoupler[0] 	:= 0;
// aStartPointCoupler[1] 	:= 0;
// aEndPointCoupler[0]		:= 0;
// aEndPointCoupler[1]		:= 100;

//Start values FOR 81984
// aStartPointCoupler[0] 	:= 0;
// aStartPointCoupler[1] 	:= 0;
// aEndPointCoupler[0]		:= 0;
// aEndPointCoupler[1]		:= 100;

eAlgorithm 		:= TCVN_EDA_APPROX_ERF;

bSuccess_ImageTransform	:= FALSE ;
bSuccess_LeftLocate		:= FALSE ;
bSuccess_RightLocate	:= FALSE ;
bSuccess_DrawCircle		:= FALSE ;
bSuccess_FindEllipse	:= FALSE ;
bGreatSuccess := FALSE;

hr := F_VN_ConvertColorSpace(ipSrcImage:= ImageRaw , ipDestImage:= ipImageProsessed ,
eTransform:= ETcVnColorSpaceTransform.TCVN_CST_GRAY_TO_RGB, hrPrev:= hr);	
bSuccess_ImageTransform := SUCCEEDED(hr);


IF bModeFixtureToGripper THEN
	// Left Claw positioning
	hr := F_VN_LocateEdgeExp(
		ipSrcImage:= ImageRaw, 
		ipEdgePoints:= ipEdgePointsL, 
		aStartPoint:= aStartPoint1, 
		aEndPoint:= aEndPoint1, 
		eEdgeDirection:= TCVN_ED_DARK_TO_LIGHT, 
		fMinStrength:= 120,
		fSearchLineDist  := 10,
		nMaxThickness := 20,
		nSearchLines:= 31,
		eAlgorithm := eAlgorithm,
		nSubpixelsIterations := 10,
		fApproxPrecision := 0.001,
		hrPrev:= hr, 
		fAvgStrength=> fFoundStr);
	bSuccess_LeftLocate := SUCCEEDED(hr);
	IF SUCCEEDED(hr) THEN
		hr := F_VN_GetAt_TcVnVector2_REAL(ipContainer:= ipEdgePointsL, aElement:= aElement1, nIndex:= 0, hrPrev:= hr);
		hr := F_VN_DrawPoints(
			ipPoints:= ipEdgePointsL, 
			ipDestImage:= ipImageProsessed, 
			eShape:= ETcVnDrawShape.TCVN_DS_X, 
			aColor:= Color.Lime, 
			hrPrev:= hr);
		hr := F_VN_FitLine(
			ipPointSet 	:= ipEdgePointsL, 
			hrPrev		:= hr,
			aFitLine	:= aFitlineL);
		hr := F_VN_DrawLine_TcVnVector4_LREAL(
			ipDestImage := ipImageProsessed,
			aColor		:= Color.Aqua,
			nThickness	:= 1,
			aLine		:= aFitlineL,
			hrPrev		:= hr);
		rClawLLineAngleRad := ATAN(aFitlineL[0]/ aFitlineL[1]); 	
 		rClawLLineAngleDeg := rClawLLineAngleRad * (180/PI); 
// 		IF rClawLLineAngleDeg > 0 THEN
// 			rClawLLineAngleDeg := rClawLLineAngleDeg - 90;
// 		ELSE
// 			rClawLLineAngleDeg := -rClawLLineAngleDeg - 90;
// 		END_IF
	END_IF
	
	// Right Claw positioning
	hr := F_VN_LocateEdgeExp(
		ipSrcImage:= ImageRaw, 
		ipEdgePoints:= ipEdgePointsR, 
		aStartPoint:= aStartPoint2, 
		aEndPoint:= aEndPoint2, 
		eEdgeDirection:= TCVN_ED_DARK_TO_LIGHT, 
		fMinStrength:= 120,
		fSearchLineDist  := 10,
		nMaxThickness := 20,
		nSearchLines:= 31,
		eAlgorithm := eAlgorithm,
		nSubpixelsIterations := 10,
		fApproxPrecision := 0.001,
		hrPrev:= hr, 
		fAvgStrength=> fFoundStr);
	bSuccess_RightLocate := SUCCEEDED(hr);
	IF SUCCEEDED(hr) THEN
		hr := F_VN_GetAt_TcVnVector2_REAL(ipContainer:= ipEdgePointsR, aElement:= aElement2, nIndex:= 0, hrPrev:= hr);
		hr := F_VN_DrawPoints(
			ipPoints:= ipEdgePointsR, 
			ipDestImage:= ipImageProsessed, 
			eShape:= ETcVnDrawShape.TCVN_DS_X, 
			aColor:= Color.Lime, 
			hrPrev:= hr);
		hr := F_VN_FitLine(
			ipPointSet 	:= ipEdgePointsR, 
			hrPrev		:= hr,
			aFitLine	:= aFitlineR);
		hr := F_VN_DrawLine_TcVnVector4_LREAL(
			ipDestImage := ipImageProsessed,
			aColor		:= Color.Aqua,
			nThickness	:= 1,
			aLine		:= aFitlineR,
			hrPrev		:= hr);
		rClawRLineAngleRad := ATAN(aFitlineR[0]/ aFitlineR[1]); 	
		rClawRLineAngleDeg := rClawRLineAngleRad * (180/PI); 
// 		IF rClawRLineAngleDeg > 0 THEN
// 			rClawRLineAngleDeg := rClawRLineAngleDeg - 90;
// 		ELSE
// 			rClawRLineAngleDeg := -rClawRLineAngleDeg - 90;
// 		END_IF
	END_IF
END_IF


hr := F_VN_DrawCircle(
		nCenterX 	:= REAL_TO_UDINT(aCenter[0]),
		nCenterY	:= REAL_TO_UDINT(aCenter[1]),
		nRadius		:= REAL_TO_UDINT(fTargetRadius),
		ipDestImage	:= ipImageProsessed,
		aColor		:= Color.Aqua,
		nThickness	:= 1,
		hrPrev		:= hr
);
bSuccess_DrawCircle := SUCCEEDED(hr);
// Circle Finding (voi laittaa joko fixturoituna gripperiin tai jos robotin paikka tarpeeksi vakio, keskiö kovakoodattuna)
IF rThreshold > 1 THEN
	hr := F_VN_Threshold(
		ipSrcImage      :=  ImageRaw,
		ipDestImage     :=  ImageFilter,
		fThreshold      :=  rThreshold, // half value range: (2^8)/2=128
		fMaxValue       :=  rMaxvalue, // max value of 8-bit image: (2^8)-1=255
		eThresholdType  :=  TCVN_TT_BINARY,
		hrPrev          :=  hr
	);
ELSE
	hr := F_VN_CopyImage(ipSrcImage := ImageRaw, ipDestImage := ImageFilter, hrPrev := hr);
END_IF
hr := F_VN_CopyIntoDisplayableImage (ImageFilter, ImageFilterDisp, hr);
hr := F_VN_LocateEllipseExp(
	ipSrcImage				:= ImageRaw, 
	ipContourPoints			:= ipEdgePointsR, 
	aCenter					:= aCenter,  
	eEdgeDirection			:= TCVN_ED_DARK_TO_LIGHT, 
	fMinStrength			:= 30, // 30
	hrPrev 					:= hr,
	fMinSearchRadius 		:= fMinRadius,
	fSearchRadius 			:= fTargetRadius,
	eAlgorithm				:= eAlgorithm,
	nSubpixelsIterations	:= 10,
	fApproxPrecision		:= 0.001,
	nMaxThickness			:= 10,
	nSearchLines			:= 31,
	bInvertSearchDirection	:= TRUE,
	stEllipse				:= stMotorEllipse
);
bSuccess_FindEllipse := SUCCEEDED(hr);
IF SUCCEEDED(hr) THEN
	
//  	hr :=  F_VN_DrawPoints(
// 		ipPoints:= ipContourPoints, 
// 		ipDestImage:= ipImageProsessed, 
// 		eShape:= ETcVnDrawShape.TCVN_DS_X, 
// 		aColor:= Color.Lime, 
// 		hrPrev:= hr);
	hr := F_VN_DrawEllipse(
		hrPrev		:= hr,
		stEllipse 	:= stMotorEllipse,
		ipDestImage := ipImageProsessed,
		aColor		:= Color.Lime,
		nThickness	:= 1,	
	);
	hr := F_VN_DrawPoint(
		nX 			:= REAL_TO_UDINT(stMotorEllipse.aCenter[0]),
		nY			:= REAL_TO_UDINT(stMotorEllipse.aCenter[1]),
		ipDestImage := ipImageProsessed,
		aColor		:= Color.Lime,
		eShape		:= ETcVnDrawShape.TCVN_DS_CIRCLE,
		hrPrev		:= hr);
END_IF

// Tähän vielä couplerin viivanhaku löydetyn ellipsin keskipisteen perusteella.

aStartPointCoupler[0] := aStartPointCoupler[0] + stMotorEllipse.aCenter[0];
aStartPointCoupler[1] := aStartPointCoupler[1] + stMotorEllipse.aCenter[1];
aEndPointCoupler[0] := aEndPointCoupler[0] + stMotorEllipse.aCenter[0];
aEndPointCoupler[1] := aEndPointCoupler[1] + stMotorEllipse.aCenter[1];

hr := F_VN_DrawPoint(
		nX 			:= REAL_TO_UDINT(aStartPointCoupler[0]),
		nY			:= REAL_TO_UDINT(aStartPointCoupler[1]),
		ipDestImage := ipImageProsessed,
		aColor		:= Color.Red,
		eShape		:= ETcVnDrawShape.TCVN_DS_SQUARE,
		hrPrev		:= hr);
		
hr := F_VN_DrawPoint(
		nX 			:= REAL_TO_UDINT(aEndPointCoupler[0]),
		nY			:= REAL_TO_UDINT(aEndPointCoupler[1]),
		ipDestImage := ipImageProsessed,
		aColor		:= Color.Red,
		eShape		:= ETcVnDrawShape.TCVN_DS_DIAMOND,
		hrPrev		:= hr);

hr := F_VN_LocateEdgeExp(
	ipSrcImage:= ImageFilter, 
	ipEdgePoints:= ipEdgePointsR, 
	aStartPoint:= aStartPointCoupler,
	aEndPoint:= aEndPointCoupler, 
	eEdgeDirection:= TCVN_ED_LIGHT_TO_DARK, 
	fMinStrength:= 100,
	fSearchLineDist  := rSearchLineDist,
	nMaxThickness := 10,
	nSearchLines:= 10,
	eAlgorithm := eAlgorithm,
	nSubpixelsIterations := 10,
	fApproxPrecision := 0.001,
	hrPrev:= hr, 
	fAvgStrength=> fFoundStr);
bGreatSuccess := SUCCEEDED(hr);
IF SUCCEEDED(hr) THEN
	FOR i := 1 TO 10 DO
		hr := F_VN_GetAt_TcVnVector2_REAL(ipContainer:= ipEdgePointsR, aElement:= aElement2, nIndex:= i, hrPrev:= hr);
		x[i] := aElement2[0];
		y[i] := aElement2[1];
	END_FOR 
	RMSE(x := x, y := y,bExecute := TRUE);
	hr := F_VN_GetAt_TcVnVector2_REAL(ipContainer:= ipEdgePointsR, aElement:= aElement2, nIndex:= 0, hrPrev:= hr);
	hr := F_VN_DrawPoints(
		ipPoints:= ipEdgePointsR, 
		ipDestImage:= ipImageProsessed, 
		eShape:= ETcVnDrawShape.TCVN_DS_X, 
		aColor:= Color.Lime, 
		hrPrev:= hr);
	hr := F_VN_FitLine(
		ipPointSet 	:= ipEdgePointsR, 
		hrPrev		:= hr,
		aFitLine	:= aFitlineR);
		
		
	rLineAngleRad := ATAN(aFitlineR[0]/ aFitlineR[1]); 	
	rLineAngleDeg := rLineAngleRad * (180/PI);
	IF rLineAngleDeg > 0 THEN
		rLineAngleDeg := rLineAngleDeg - 90;
	ELSE
		rLineAngleDeg := -rLineAngleDeg - 90;
	END_IF
	rLineAngleResultDeg :=  rLineAngleDeg + ((rClawRLineAngleDeg + rClawLLineAngleDeg)/2);
	IF NOT bRmsErr THEN
		IF rLineAngleResultDeg < 10  AND rLineAngleResultDeg > -10 THEN
			stCouplerData.rCouplerAngleDeg := rLineAngleResultDeg;
			stCouplerData.rCouplerAngleRad := (rLineAngleResultDeg * (PI/180));
			stCouplerData.bPartDetectFailed := FALSE;
			stCouplerData.bPartDetectSucceeded := TRUE;
		ELSE
			stCouplerData.bPartDetectSucceeded := FALSE;
			stCouplerData.bPartDetectFailed := TRUE;
		END_IF
	ELSE
		stCouplerData.bPartDetectSucceeded := FALSE;
		stCouplerData.bPartDetectFailed := TRUE;
	END_IF
	hr := F_VN_DrawLine_TcVnVector4_LREAL(
		ipDestImage := ipImageProsessed,
		aColor		:= Color.Aqua,
		nThickness	:= 1,
		aLine		:= aFitlineR,
		hrPrev		:= hr);
END_IF
END_METHOD

METHOD PositionDetect : BOOL

VAR
	EdgeLoop 					: ULINT;
	nNewArrayValue 				: INT;
	
	bCheckOnce 					: BOOL := TRUE;
	bCheckOnceSuc				: BOOL := TRUE;
	
	aStartPointT 				: TcVnPoint2_REAL;
	aEndPointT					: TcVnPoint2_REAL;
	aStartPointS 				: TcVnPoint2_REAL;
	aEndPointS					: TcVnPoint2_REAL;
	
	ipEdgePointsT				: ITcVnContainer;
	ipEdgePointsS				: ITcVnContainer;
	hrEdgeT						: HRESULT;

	EdgeLoopDown 					: ULINT;
	EndPointXTDown 					: REAL := 0;
	aElementTopDown 				: TcVnPoint2_REAL;
	nNewArrayValueDown 				: INT;
	
	
	aStartPointTDown 				: TcVnPoint2_REAL;
	aEndPointTDown					: TcVnPoint2_REAL;
	ipEdgePointsTDown				: ITcVnContainer;
	aLine           				: TcVnVector4_LREAL;


	PartAnglerad					: LREAL;
	PartAngle						: LREAL;
	EndPointXT 						: REAL := 0;
	nOffset							: INT;
	nPixelMax						: LREAL := 10;
	
END_VAR
EndPointXT := 0;
hrEdgeT := 0;


hrEdgeT := F_VN_LocateEdge(
	ipSrcImage:= ImageRaw, 
	ipEdgePoints:= ipEdgePointsT, 
	aStartPoint:= aStartPointT, 
	aEndPoint:= aEndPointT, 
	eEdgeDirection:= ETcVnEdgeDirection.TCVN_ED_Light_TO_Dark, 
	fMinStrength:= 45, 
	nSearchLines:= 1, 
	hrPrev:= hr, 
	fAvgStrength=> );
hrEdgeT := F_VN_LocateEdge(
	ipSrcImage:= ImageRaw, 
	ipEdgePoints:= ipEdgePointsS, 
	aStartPoint:= aStartPointS, 
	aEndPoint:= aEndPointS, 
	eEdgeDirection:= ETcVnEdgeDirection.TCVN_ED_Light_TO_Dark, 
	fMinStrength:= 45, 
	nSearchLines:= 1, 
	hrPrev:= hr, 
	fAvgStrength=> );
IF SUCCEEDED(hrEdgeT) THEN
	hrEdgeT := F_VN_DrawPoints(
		ipPoints:= ipEdgePointsT, 
		ipDestImage:= ipImageProsessed, 
		eShape:= ETcVnDrawShape.TCVN_DS_X, 
		aColor:= Color.Lime, 
		hrPrev:= hr);
	hrEdgeT := F_VN_GetAt_TcVnVector2_REAL(ipContainer:= ipEdgePointsT, aElement:= aElement1, nIndex:= 0, hrPrev:= hrEdgeT);
	hrEdgeT := F_VN_GetAt_TcVnVector2_REAL(ipContainer:= ipEdgePointsS, aElement:= aElement2, nIndex:= 0, hrPrev:= hrEdgeT);
ELSE
	IF bCheckOnce THEN
		ADSLOGSTR(msgCtrlMask := ADSLOG_MSGTYPE_ERROR, msgFmtStr := 'Error1', strArg:= ' ');
		bCheckOnce := FALSE;
	END_IF
	EndPointXT := EndPointXT + 30;
END_IF
END_METHOD

METHOD RMSE : BOOL
VAR_INPUT // This method calculates the RMS Error value of found points
    x : ARRAY[1..10] OF LREAL;
    y : ARRAY[1..10] OF LREAL;
	bExecute : BOOL;
END_VAR
VAR
 	i       : INT;
    n       : LREAL := 10.0;
    sumX    : LREAL := 0.0;
    sumY    : LREAL := 0.0;
    sumXY   : LREAL := 0.0;
    sumX2   : LREAL := 0.0;
    yFit    : LREAL;
    errSum  : LREAL := 0.0;	

END_VAR
sumX := 0;
sumY := 0;
sumXY := 0;
sumX2 := 0;
IF bExecute THEN
	FOR i := 1 TO 10 DO
		sumX  := sumX  + x[i];
		sumY  := sumY  + y[i];
		sumXY := sumXY + (x[i] * y[i]);
		sumX2 := sumX2 + (x[i] * x[i]);
	END_FOR
	
	
	IF (n * sumX2 - sumX * sumX) <> 0 THEN
		slope := (n * sumXY - sumX * sumY) /
				 (n * sumX2 - sumX * sumX);
	ELSE
		slope := 0;
	END_IF
	intercept := (sumY - slope * sumX) / n;
	FOR i := 1 TO 10 DO
		yFit := slope * x[i] + intercept;
		errSum := errSum + (y[i] - yFit) * (y[i] - yFit);
	END_FOR
	
	rmsError := SQRT(errSum / n);
	IF rmsError > 1.5 THEN
		bRmsErr := TRUE;
	ELSE
		bRmsErr := FALSE;
	END_IF
	bExecute := FALSE;
END_IF
END_METHOD

METHOD SetParams : BOOL
VAR_INPUT
END_VAR
CASE iStationId OF
	1..5:
		rThreshold := stRecipeData.Station1To5.rThreshold;
		aStartPointCoupler := stRecipeData.Station1To5.aStartPointCoupler;
		aEndPointCoupler := stRecipeData.Station1To5.aEndPointCoupler;
		rSearchLineDist :=  stRecipeData.Station1To5.rSearchLineDist;
	6..10:
		rThreshold := stRecipeData.Station5To10.rThreshold;
		aStartPointCoupler := stRecipeData.Station5To10.aStartPointCoupler;
		aEndPointCoupler := stRecipeData.Station5To10.aEndPointCoupler;
		rSearchLineDist :=  stRecipeData.Station5To10.rSearchLineDist;
END_CASE
END_METHOD

METHOD TrigImage : BOOL
VAR_INPUT
END_VAR
fbCamera.TriggerImage();
END_METHOD

END_FUNCTION_BLOCK

// ---- POUs/VisMain/FB_InfeedCam.TcPOU
FUNCTION_BLOCK FB_InfeedCam
VAR_INPUT
	bTriggerImage : BOOL;
 	stPosData : REFERENCE TO ST_PalletImagingData;
 	stImagingSetValues : REFERENCE TO ST_Recipes;
	bDetectPallet1To5 : BOOL;
	bDetectPallet6To10 : BOOL;
END_VAR
VAR_OUTPUT
	bImageReceived : BOOL;
	bPartDetectFailed : BOOL;
	bDone : BOOL;
END_VAR
VAR
	hr									: HRESULT;
	eVisionState						: ETcVnCameraState;
	fbCamera          					: FB_VN_GevCameraControl;
	ImageRawDisp						: ITcVnDisplayableImage;
	ImageFilter							: Tc3_Vision.ITcVnImage;
	ImageFilterDisp						: ITcVnDisplayableImage;
	nNewImageCounter 					: UINT;
	ImageRaw							: Tc3_Vision.ITcVnImage;
	ImageProsessed						: Tc3_Vision.ITcVnImage;
	ipImageTest							: ITcVnImage;
	ipImageTestDisp						: ITcVnDisplayableImage;
	
	stRectangle							: TcVnRotatedRectangle;
	ImageProsessedDisp					: Tc3_Vision.ITcVnDisplayableImage;
	

	rThreshold			: LREAL := 20;
	rMaxvalue			: LREAL := 255;
	
	fFoundStr : REAL;
	eAlgorithm           				: ETcVnEdgeDetectionAlgorithm;
	aStartPoint1 						: TcVnPoint2_REAL;
	aEndPoint1							: TcVnPoint2_REAL;
	ipEdgePointsL    					: ITcVnContainer;
	aFitlineL							: TcVnVector4_LREAL;
	aElement1 							: TcVnPoint2_REAL;
	
	aStartPoint2 						: TcVnPoint2_REAL;
	aEndPoint2							: TcVnPoint2_REAL;
	ipEdgePoints14mm    				: ITcVnContainer;
	aFitline2							: TcVnVector4_LREAL;
	aElement2 							: TcVnPoint2_REAL;
	
	aStartPoint3 						: TcVnPoint2_REAL;
	aEndPoint3							: TcVnPoint2_REAL;
	ipEdgePoints3	    				: ITcVnContainer;
	aFitline3							: TcVnVector4_LREAL;
	aElement3 							: TcVnPoint2_REAL;
	
	aStartPointMirr1 						: TcVnPoint2_REAL;
	aEndPointMirr1							: TcVnPoint2_REAL;
	ipEdgePointsMirr1    					: ITcVnContainer;
	
	aStartPointMirr2 						: TcVnPoint2_REAL;
	aEndPointMirr2							: TcVnPoint2_REAL;
	ipEdgePointsMirr2   					: ITcVnContainer;
	
	stDetectionArea1							: TcVnRectangle_UDINT;
	stDetectionArea2							: TcVnRectangle_UDINT;
	aAverage  							: TcVnVector4_LREAL;
	aStdDev								: TcVnVector4_LREAL;
	aSavedStdDev						: ARRAY [0..4] OF LREAL;
	aPalletBinary						: ARRAY [0..5] OF BOOL;
	wPalletBinary1						: WORD;
	wPalletBinary2						: WORD;
	iDetectPos 							: INT;
END_VAR

eVisionState := fbCamera.GetState();
eAlgorithm 		:= TCVN_EDA_APPROX_ERF;


IF stImagingSetValues.Station1To5.rGalvoThickness = 9.5 THEN
	stPosData.bTogglePallet := TRUE;
ELSIF stImagingSetValues.Station1To5.rGalvoThickness = 14 THEN	
	stPosData.bTogglePallet := FALSE;
END_IF

SetPoints();

IF eVisionState = TCVN_CS_ERROR THEN
	hr := fbCamera.Reset();
ELSIF eVisionState = TCVN_CS_TRIGGERING THEN
	hr := fbCamera.TriggerImage();
ELSIF eVisionState < TCVN_CS_ACQUIRING THEN
    hr := fbCamera.StartAcquisition();
ELSIF eVisionState = TCVN_CS_ACQUIRING THEN
	hr := fbCamera.GetCurrentImageUndistorted(ImageRaw); // switch to undistorted
	IF SUCCEEDED(hr) AND ImageRaw <> 0 THEN
		stPosData.bSuccess_10mmLocate := FALSE;
		stPosData.bSuccess_14mmLocate := FALSE;
		nNewImageCounter := nNewImageCounter +1;
		bPartDetectFailed := FALSE;
		bImageReceived := TRUE;
		hr := F_VN_CopyIntoDisplayableImage (ImageRaw, ImageRawDisp, hr);
		GalvoPalletDetect();
		MirrorPalletDetect();
	END_IF
END_IF

METHOD GalvoPalletDetect : BOOL
VAR_INPUT
END_VAR

hr := F_VN_Threshold(
	ipSrcImage      :=  ImageRaw,
	ipDestImage     :=  ImageFilter,
	fThreshold      :=  rThreshold, // half value range: (2^8)/2=128
	fMaxValue       :=  rMaxvalue, // max value of 8-bit image: (2^8)-1=255
	eThresholdType  :=  TCVN_TT_BINARY,
	hrPrev          :=  hr);
hr := F_VN_CopyIntoDisplayableImage (ImageFilter, ImageFilterDisp, hr);
hr := F_VN_ConvertColorSpace(ipSrcImage:= ImageRaw , ipDestImage:= ImageProsessed ,
eTransform:= ETcVnColorSpaceTransform.TCVN_CST_GRAY_TO_RGB, hrPrev:= hr);	
IF stPosData.bTogglePallet THEN	
	hr := F_VN_LocateEdgeExp(
		ipSrcImage:= ImageRaw, 
		ipEdgePoints:= ipEdgePointsL, 
		aStartPoint:= aStartPoint1, 
		aEndPoint:= aEndPoint1, 
		eEdgeDirection:= TCVN_ED_DARK_TO_LIGHT, 
		fMinStrength:= 60,
		fSearchLineDist  := 10,
		nMaxThickness := 20,
		nSearchLines:= 10,
		eAlgorithm := eAlgorithm,
		nSubpixelsIterations := 10,
		fApproxPrecision := 0.001,
		hrPrev:= hr, 
		fAvgStrength=> fFoundStr);
stPosData.bSuccess_10mmLocate := SUCCEEDED(hr);
	IF SUCCEEDED(hr) THEN
		hr := F_VN_GetAt_TcVnVector2_REAL(ipContainer:= ipEdgePointsL, aElement:= aElement1, nIndex:= 0, hrPrev:= hr);
		hr := F_VN_DrawPoints(
			ipPoints:= ipEdgePointsL, 
			ipDestImage:= ImageProsessed, 
			eShape:= ETcVnDrawShape.TCVN_DS_X, 
			aColor:= Color.Lime, 
			hrPrev:= hr);
		hr := F_VN_FitLine(
			ipPointSet 	:= ipEdgePointsL, 
			hrPrev		:= hr,
			aFitLine	:= aFitlineL);
		hr := F_VN_DrawLine_TcVnVector4_LREAL(
			ipDestImage := ImageProsessed,
			aColor		:= Color.Aqua,
			nThickness	:= 1,
			aLine		:= aFitlineL,
			hrPrev		:= hr);
	
		hr := F_VN_CopyIntoDisplayableImage (ImageProsessed, ImageProsessedDisp, hr);
	END_IF
ELSE
	hr := F_VN_LocateEdgeExp(
		ipSrcImage:= ImageRaw, 
		ipEdgePoints:= ipEdgePoints14mm, 
		aStartPoint:= aStartPoint2, 
		aEndPoint:= aEndPoint2, 
		eEdgeDirection:= TCVN_ED_LIGHT_TO_DARK, 
		fMinStrength:= 45,
		fSearchLineDist  := 10,
		nMaxThickness := 20,
		nSearchLines:= 5,
		eAlgorithm := eAlgorithm,
		nSubpixelsIterations := 10,
		fApproxPrecision := 0.001,
		hrPrev:= hr, 
		fAvgStrength=> fFoundStr);
	stPosData.bSuccess_14mmLocate := SUCCEEDED(hr);
	IF SUCCEEDED(hr) THEN
		hr := F_VN_GetAt_TcVnVector2_REAL(ipContainer:= ipEdgePoints14mm, aElement:= aElement1, nIndex:= 0, hrPrev:= hr);
		hr := F_VN_DrawPoints(
			ipPoints:= ipEdgePoints14mm, 
			ipDestImage:= ImageProsessed, 
			eShape:= ETcVnDrawShape.TCVN_DS_X, 
			aColor:= Color.Lime, 
			hrPrev:= hr);
		hr := F_VN_FitLine(
			ipPointSet 	:= ipEdgePoints14mm, 
			hrPrev		:= hr,
			aFitLine	:= aFitline2);
		hr := F_VN_DrawLine_TcVnVector4_LREAL(
			ipDestImage := ImageProsessed,
			aColor		:= Color.Aqua,
			nThickness	:= 1,
			aLine		:= aFitline2,
			hrPrev		:= hr);
		hr := F_VN_CopyIntoDisplayableImage (ImageProsessed, ImageProsessedDisp, hr);
	END_IF
	hr := F_VN_LocateEdgeExp(
		ipSrcImage:= ImageRaw, 
		ipEdgePoints:= ipEdgePoints3, 
		aStartPoint:= aStartPoint3, 
		aEndPoint:= aEndPoint3, 
		eEdgeDirection:= TCVN_ED_LIGHT_TO_DARK, 
		fMinStrength:= 45,
		fSearchLineDist  := 10,
		nMaxThickness := 20,
		nSearchLines:= 5,
		eAlgorithm := eAlgorithm,
		nSubpixelsIterations := 10,
		fApproxPrecision := 0.001,
		hrPrev:= hr, 
		fAvgStrength=> fFoundStr);
	stPosData.bSuccess_14mmLocate := SUCCEEDED(hr);
	IF SUCCEEDED(hr) THEN
		hr := F_VN_GetAt_TcVnVector2_REAL(ipContainer:= ipEdgePoints3, aElement:= aElement3, nIndex:= 0, hrPrev:= hr);
		hr := F_VN_DrawPoints(
			ipPoints:= ipEdgePoints3, 
			ipDestImage:= ImageProsessed, 
			eShape:= ETcVnDrawShape.TCVN_DS_X, 
			aColor:= Color.Lime, 
			hrPrev:= hr);
		hr := F_VN_FitLine(
			ipPointSet 	:= ipEdgePoints3, 
			hrPrev		:= hr,
			aFitLine	:= aFitline3);
		hr := F_VN_DrawLine_TcVnVector4_LREAL(
			ipDestImage := ImageProsessed,
			aColor		:= Color.Aqua,
			nThickness	:= 1,
			aLine		:= aFitline3,
			hrPrev		:= hr);
		hr := F_VN_CopyIntoDisplayableImage (ImageProsessed, ImageProsessedDisp, hr);
	END_IF
END_IF
END_METHOD

METHOD MirrorPalletDetect : BOOL
VAR_INPUT
END_VAR
VAR
	
END_VAR
stDetectionArea1.nHeight := 8;
stDetectionArea1.nWidth := 10;
stDetectionArea1.nX := 90;
stDetectionArea1.nY := 27;
iDetectPos := 0;

stDetectionArea2.nHeight := 8;
stDetectionArea2.nWidth := 10;
stDetectionArea2.nX := 631;
stDetectionArea2.nY := 27;
hr := F_VN_CopyImage(ImageRaw, ipImageTest, hrPrev := hr);
hr:= F_VN_ConvertColorSpace(ipSrcImage:= ipImageTest , ipDestImage:= ipImageTest ,
		eTransform:= ETcVnColorSpaceTransform.TCVN_CST_GRAY_TO_RGB, hrPrev:= hr);
IF bDetectPallet1To5 THEN
	hr := F_VN_LocateEdgeExp(
		ipSrcImage:= ImageRaw, 
		ipEdgePoints:= ipEdgePointsMirr1, 
		aStartPoint:= aStartPointMirr1, 
		aEndPoint:= aEndPointMirr1, 
		eEdgeDirection:= TCVN_ED_LIGHT_TO_DARK, 
		fMinStrength:= 45,
		fSearchLineDist  := 10,
		nMaxThickness := 20,
		nSearchLines:= 5,
		eAlgorithm := eAlgorithm,
		nSubpixelsIterations := 10,
		fApproxPrecision := 0.001,
		hrPrev:= hr, 
		fAvgStrength=> );
	IF Succeeded(hr) THEN
		hr := F_VN_SetRoi_TcVnRectangle_UDINT(stRoi:= stDetectionArea1, ipDestImage:= ipImageTest, hrPrev:= hr);
		hr := F_VN_ImageAverageStdDev(ipSrcImage:= ipImageTest,aStdDev := aStdDev, aAverage:= aAverage, hrPrev:= hr);
		hr := F_VN_ResetRoi(ipImage:= ipImageTest, hrPrev:= hr);
		hr := F_VN_DrawRectangle_TcVnRectangle_UDINT(
			stRectangle:= stDetectionArea1,
			ipDestImage:= ipImageTest,
			aColor:= Color.Green,
			nThickness:= 1,
			hrPrev:= hr);
		IF aStdDev[0] > 20 THEN
			wPalletBinary1 := wPalletBinary1 OR SHL(1, 0);
		ELSE
			wPalletBinary1 := wPalletBinary1 AND NOT SHL(1, 0);
		END_IF
		stDetectionArea1.nY := stDetectionArea1.nY + 22;
		FOR iDetectPos := 1 TO 4 DO
			hr := F_VN_SetRoi_TcVnRectangle_UDINT(stRoi:= stDetectionArea1, ipDestImage:= ipImageTest, hrPrev:= hr);
// 			hr := F_VN_ImageAverage(ipSrcImage:= ipImageTest, aAverage:= aAverage, hrPrev:= hr);
			hr := F_VN_ImageAverageStdDev(ipSrcImage:= ipImageTest,aStdDev := aStdDev, aAverage:= aAverage, hrPrev:= hr);
			hr := F_VN_ResetRoi(ipImage:= ipImageTest, hrPrev:= hr);
			hr := F_VN_DrawRectangle_TcVnRectangle_UDINT(
				stRectangle:= stDetectionArea1,
				ipDestImage:= ipImageTest,
				aColor:= Color.Green,
				nThickness:= 1,
				hrPrev:= hr);
			IF aAverage[0] > 160 THEN
				wPalletBinary1 := wPalletBinary1 OR SHL(1, iDetectPos);
			ELSE
				wPalletBinary1 := wPalletBinary1 AND NOT SHL(1, iDetectPos);
			END_IF
			IF iDetectPos = 1 THEN
				stDetectionArea1.nY := stDetectionArea1.nY + 98;
			ELSE
				stDetectionArea1.nY := stDetectionArea1.nY + 21;
			END_IF
			aSavedStdDev[iDetectPos] := aStdDev[0];
		END_FOR
		IF SUCCEEDED(hr) THEN
			hr := F_VN_CopyIntoDisplayableImage (ipImageTest, ipImageTestDisp, hr);	
		END_IF
		bDetectPallet1To5 := FALSE;
	ELSE
		// ERROR 402
		Err.Err;
	END_IF
END_IF
IF bDetectPallet6To10 THEN
	hr := F_VN_LocateEdgeExp(
		ipSrcImage:= ImageRaw, 
		ipEdgePoints:= ipEdgePointsMirr2, 
		aStartPoint:= aStartPointMirr2, 
		aEndPoint:= aEndPointMirr2, 
		eEdgeDirection:= TCVN_ED_LIGHT_TO_DARK, 
		fMinStrength:= 45,
		fSearchLineDist  := 10,
		nMaxThickness := 20,
		nSearchLines:= 5,
		eAlgorithm := eAlgorithm,
		nSubpixelsIterations := 10,
		fApproxPrecision := 0.001,
		hrPrev:= hr, 
		fAvgStrength=> );
	IF Succeeded(hr) THEN
		FOR iDetectPos := 0 TO 1 DO
			hr := F_VN_SetRoi_TcVnRectangle_UDINT(stRoi:= stDetectionArea2, ipDestImage:= ipImageTest, hrPrev:= hr);
			hr := F_VN_ImageAverageStdDev(ipSrcImage:= ipImageTest,aStdDev := aStdDev, aAverage:= aAverage, hrPrev:= hr);
			hr := F_VN_ResetRoi(ipImage:= ipImageTest, hrPrev:= hr);
			hr := F_VN_DrawRectangle_TcVnRectangle_UDINT(
				stRectangle:= stDetectionArea2,
				ipDestImage:= ipImageTest,
				aColor:= Color.Green,
				nThickness:= 1,
				hrPrev:= hr);
			IF aStdDev[0] > 20 THEN
				wPalletBinary2 := wPalletBinary2 OR SHL(1, 0);
			ELSE
				wPalletBinary2 := wPalletBinary2 AND NOT SHL(1, 0);
			END_IF
			stDetectionArea2.nY := stDetectionArea2.nY + 22;
		END_FOR
		FOR iDetectPos := 2 TO 4 DO
			hr := F_VN_SetRoi_TcVnRectangle_UDINT(stRoi:= stDetectionArea2, ipDestImage:= ipImageTest, hrPrev:= hr);
// 			hr := F_VN_ImageAverage(ipSrcImage:= ipImageTest, aAverage:= aAverage, hrPrev:= hr);
			hr := F_VN_ImageAverageStdDev(ipSrcImage:= ipImageTest,aStdDev := aStdDev, aAverage:= aAverage, hrPrev:= hr);
			hr := F_VN_ResetRoi(ipImage:= ipImageTest, hrPrev:= hr);
			hr := F_VN_DrawRectangle_TcVnRectangle_UDINT(
				stRectangle:= stDetectionArea2,
				ipDestImage:= ipImageTest,
				aColor:= Color.Green,
				nThickness:= 1,
				hrPrev:= hr);
			IF aAverage[0] > 160 THEN
				wPalletBinary2 := wPalletBinary2 OR SHL(1, iDetectPos);
			ELSE
				wPalletBinary2 := wPalletBinary2 AND NOT SHL(1, iDetectPos);
			END_IF
			IF iDetectPos = 1 THEN
				stDetectionArea2.nY := stDetectionArea2.nY + 98;
			ELSE
				stDetectionArea2.nY := stDetectionArea2.nY + 21;
			END_IF
			aSavedStdDev[iDetectPos] := aStdDev[0];
		END_FOR
		IF SUCCEEDED(hr) THEN
			hr := F_VN_CopyIntoDisplayableImage (ipImageTest, ipImageTestDisp, hr);	
		END_IF
		bDetectPallet6To10 := FALSE;
	ELSE
		// ERROR 402
		Err.Err;
	END_IF
END_IF
END_METHOD

ACTION SetPoints:
aStartPoint1[0] := 1100;
aStartPoint1[1] := 730;
aEndPoint1[0] 	:= 1100;
aEndPoint1[1] 	:= 770;


aStartPoint2[0] := 1;
aStartPoint2[1] := 530;
aEndPoint2[0] 	:= 50;
aEndPoint2[1] 	:= 530;

aStartPoint3[0] := 1140;
aStartPoint3[1] := 530;
aEndPoint3[0] 	:= 50;
aEndPoint3[1] 	:= 1040;

aStartPointMirr1[0] := 60;
aStartPointMirr1[1] := 220;
aEndPointMirr1[0] 	:= 110;
aEndPointMirr1[1] 	:= 220;

aStartPointMirr2[0] := 600;
aStartPointMirr2[1] := 220;
aEndPointMirr2[0] 	:= 660;
aEndPointMirr2[1] 	:= 220;
END_ACTION

METHOD TrigImage : BOOL
VAR_INPUT
END_VAR
fbCamera.TriggerImage();
END_METHOD

END_FUNCTION_BLOCK

// ---- POUs/VisMain/FB_OutfeedCam.TcPOU
FUNCTION_BLOCK FB_OutfeedCam
VAR_INPUT
	bCheckRow1	: BOOL;
	bCheckRow2 : BOOL;
END_VAR
VAR_OUTPUT
	bError : BOOL;
	iErrorId			: INT;
	bPalletRow1NotClear : BOOL;
	bPalletRow2NotClear : BOOL;
	bImagingDone	: BOOL;
END_VAR
VAR
	hr									: HRESULT;
	eVisionState						: ETcVnCameraState;
	fbCamera          					: FB_VN_GevCameraControl;
	ImageRawDisp						: ITcVnDisplayableImage;
	nNewImageCounter 					: UINT;
	ImageRaw: Tc3_Vision.ITcVnImage;
	ipImageTest							: ITcVnImage;
	ipImageTestDisp						: ITcVnDisplayableImage;
	
	
	stDetectionArea1					: TcVnRectangle_UDINT;
	aStdDev								: TcVnVector4_LREAL;
	aAverage  							: TcVnVector4_LREAL;
	stDetectionArea2					: TcVnRectangle_UDINT;
	aStdDev2								: TcVnVector4_LREAL;
	aAverage2  							: TcVnVector4_LREAL;
	stDetectionArea3					: TcVnRectangle_UDINT;
	aStdDev3								: TcVnVector4_LREAL;
	aAverage3  							: TcVnVector4_LREAL;
	DoneTof								: TOF;
	bInitTrig 								: BOOL;
	TrigCheckTmr							: TON;
	fbEventlogger							: FB_EventLogger;
END_VAR

eVisionState := fbCamera.GetState();
DoneTof(PT := T#0.5S, Q => bImagingDone);
DoneTof.IN := FALSE;

stDetectionArea1.nHeight := 50;
stDetectionArea1.nWidth := 1100;
stDetectionArea1.nX := 30;
stDetectionArea1.nY := 140;

stDetectionArea2.nHeight := 30;
stDetectionArea2.nWidth := 900;
stDetectionArea2.nX := 40;
stDetectionArea2.nY := 600;

stDetectionArea3.nHeight := 30;
stDetectionArea3.nWidth := 110;
stDetectionArea3.nX := 1020;
stDetectionArea3.nY := 600;

IF eVisionState = TCVN_CS_ERROR THEN
	hr := fbCamera.Reset();
ELSIF eVisionState = TCVN_CS_TRIGGERING THEN
	hr := fbCamera.TriggerImage();
ELSIF eVisionState < TCVN_CS_ACQUIRING THEN
    hr := fbCamera.StartAcquisition();
ELSIF eVisionState = TCVN_CS_ACQUIRING THEN
	hr := fbCamera.GetCurrentImage(ImageRaw); // switch to undistorted
	IF SUCCEEDED(hr) AND ImageRaw <> 0 THEN
		bError := FALSE;
		nNewImageCounter := nNewImageCounter +1;
		hr := F_VN_CopyIntoDisplayableImage (ImageRaw, ImageRawDisp, hr);
		hr := F_VN_CopyImage(ImageRaw, ipImageTest, hrPrev := hr);
		hr:= F_VN_ConvertColorSpace(ipSrcImage:= ipImageTest , ipDestImage:= ipImageTest ,
				eTransform:= ETcVnColorSpaceTransform.TCVN_CST_GRAY_TO_RGB, hrPrev:= hr);
		hr := F_VN_SetRoi_TcVnRectangle_UDINT(stRoi:= stDetectionArea1, ipDestImage:= ipImageTest, hrPrev:= hr);
		hr := F_VN_ImageAverageStdDev(ipSrcImage:= ipImageTest,aStdDev := aStdDev, aAverage:= aAverage, hrPrev:= hr);
		hr := F_VN_ResetRoi(ipImage:= ipImageTest, hrPrev:= hr);
		hr := F_VN_DrawRectangle_TcVnRectangle_UDINT(
			stRectangle:= stDetectionArea1,
			ipDestImage:= ipImageTest,
			aColor:= Color.Green,
			nThickness:= 1,
			hrPrev:= hr);
		hr := F_VN_SetRoi_TcVnRectangle_UDINT(stRoi:= stDetectionArea2, ipDestImage:= ipImageTest, hrPrev:= hr);
		hr := F_VN_ImageAverageStdDev(ipSrcImage:= ipImageTest,aStdDev := aStdDev2, aAverage:= aAverage2, hrPrev:= hr);
		hr := F_VN_ResetRoi(ipImage:= ipImageTest, hrPrev:= hr);
		hr := F_VN_DrawRectangle_TcVnRectangle_UDINT(
			stRectangle:= stDetectionArea2,
			ipDestImage:= ipImageTest,
			aColor:= Color.Green,
			nThickness:= 1,
			hrPrev:= hr);
		hr := F_VN_SetRoi_TcVnRectangle_UDINT(stRoi:= stDetectionArea3, ipDestImage:= ipImageTest, hrPrev:= hr);
		hr := F_VN_ImageAverageStdDev(ipSrcImage:= ipImageTest,aStdDev := aStdDev3, aAverage:= aAverage3, hrPrev:= hr);
		hr := F_VN_ResetRoi(ipImage:= ipImageTest, hrPrev:= hr);
		hr := F_VN_DrawRectangle_TcVnRectangle_UDINT(
			stRectangle:= stDetectionArea3,
			ipDestImage:= ipImageTest,
			aColor:= Color.Green,
			nThickness:= 1,
			hrPrev:= hr);
		IF aStdDev[0] > 13 THEN
			bPalletRow1NotClear := TRUE;
		ELSE
			bPalletRow1NotClear := FALSE;
		END_IF
		IF aStdDev3[0] > 13 OR aStdDev2[0] > 14 THEN
			bPalletRow2NotClear := TRUE;
		ELSE
			bPalletRow2NotClear := FALSE;
		END_IF
		hr := F_VN_CopyIntoDisplayableImage (ipImageTest, ipImageTestDisp, hr);
		DoneTof.IN := TRUE;
	ELSIF bInitTrig AND TrigCheckTmr.Q THEN
		bError := TRUE;
		iErrorId := 402;
		fbEventlogger.bRaiseAlarm[16]:=TRUE;
		fbEventlogger.sErrorCode:= '402';
		Err.Err;
		bInitTrig := FALSE;
		TrigCheckTmr.IN := FALSE;
	END_IF
	
END_IF

METHOD TrigImage : BOOL
VAR_INPUT
END_VAR
fbCamera.TriggerImage();
bInitTrig := TRUE;
TrigCheckTmr.IN := TRUE;
END_METHOD

END_FUNCTION_BLOCK

// ---- POUs/VisMain/FB_RejectCam.TcPOU
FUNCTION_BLOCK FB_RejectCam
VAR_INPUT
	bCheckRow1	: BOOL;
	bCheckRow2 : BOOL;
END_VAR
VAR_OUTPUT
	bError : BOOL;
	bPalletRow1NotClear : BOOL;
	bPalletRow2NotClear : BOOL;
	iErrorId			: INT;
	bImagingDone	: BOOL;
END_VAR
VAR
	hr									: HRESULT;
	eVisionState						: ETcVnCameraState;
	fbCamera          					: FB_VN_GevCameraControl;
	ImageRawDisp						: ITcVnDisplayableImage;
	nNewImageCounter 					: UINT;
	ImageRaw: Tc3_Vision.ITcVnImage;
	ipImageTest							: ITcVnImage;
	ipImageTestDisp						: ITcVnDisplayableImage;
	

	stDetectionArea1					: TcVnRectangle_UDINT;
	aStdDev								: TcVnVector4_LREAL;
	aAverage  							: TcVnVector4_LREAL;
	stDetectionArea2					: TcVnRectangle_UDINT;
	aStdDev2								: TcVnVector4_LREAL;
	aAverage2  							: TcVnVector4_LREAL;
	DoneTof								: TOF;
	bInitTrig 								: BOOL;
	TrigCheckTmr							: TON;
	fbEventlogger							: FB_EventLogger;
END_VAR

eVisionState := fbCamera.GetState();
DoneTof(PT := T#0.5S, Q => bImagingDone);
DoneTof.IN := FALSE;

stDetectionArea1.nHeight := 50;
stDetectionArea1.nWidth := 1100;
stDetectionArea1.nX := 30;
stDetectionArea1.nY := 140;

stDetectionArea2.nHeight := 25;
stDetectionArea2.nWidth := 1090;
stDetectionArea2.nX := 40;
stDetectionArea2.nY := 595;


IF eVisionState = TCVN_CS_ERROR THEN
	hr := fbCamera.Reset();
ELSIF eVisionState = TCVN_CS_TRIGGERING THEN
	hr := fbCamera.TriggerImage();
ELSIF eVisionState < TCVN_CS_ACQUIRING THEN
    hr := fbCamera.StartAcquisition();
ELSIF eVisionState = TCVN_CS_ACQUIRING THEN
	hr := fbCamera.GetCurrentImage(ImageRaw); // switch to undistorted
	IF SUCCEEDED(hr) AND ImageRaw <> 0 THEN
		bError := FALSE;
		nNewImageCounter := nNewImageCounter +1;
		hr := F_VN_CopyIntoDisplayableImage (ImageRaw, ImageRawDisp, hr);
		hr := F_VN_CopyImage(ImageRaw, ipImageTest, hrPrev := hr);
		hr:= F_VN_ConvertColorSpace(ipSrcImage:= ipImageTest , ipDestImage:= ipImageTest ,
				eTransform:= ETcVnColorSpaceTransform.TCVN_CST_GRAY_TO_RGB, hrPrev:= hr);
		hr := F_VN_SetRoi_TcVnRectangle_UDINT(stRoi:= stDetectionArea1, ipDestImage:= ipImageTest, hrPrev:= hr);
		hr := F_VN_ImageAverageStdDev(ipSrcImage:= ipImageTest,aStdDev := aStdDev, aAverage:= aAverage, hrPrev:= hr);
		hr := F_VN_ResetRoi(ipImage:= ipImageTest, hrPrev:= hr);
		hr := F_VN_DrawRectangle_TcVnRectangle_UDINT(
			stRectangle:= stDetectionArea1,
			ipDestImage:= ipImageTest,
			aColor:= Color.Green,
			nThickness:= 1,
			hrPrev:= hr);
		hr := F_VN_SetRoi_TcVnRectangle_UDINT(stRoi:= stDetectionArea2, ipDestImage:= ipImageTest, hrPrev:= hr);
		hr := F_VN_ImageAverageStdDev(ipSrcImage:= ipImageTest,aStdDev := aStdDev2, aAverage:= aAverage2, hrPrev:= hr);
		hr := F_VN_ResetRoi(ipImage:= ipImageTest, hrPrev:= hr);
		hr := F_VN_DrawRectangle_TcVnRectangle_UDINT(
			stRectangle:= stDetectionArea2,
			ipDestImage:= ipImageTest,
			aColor:= Color.Green,
			nThickness:= 1,
			hrPrev:= hr);
		IF aStdDev[0] > 13 THEN
			bPalletRow1NotClear := TRUE;
		ELSE
			bPalletRow1NotClear := FALSE;
		END_IF
		IF aStdDev2[0] > 14 THEN
			bPalletRow2NotClear := TRUE;
		ELSE
			bPalletRow2NotClear := FALSE;
		END_IF
		hr := F_VN_CopyIntoDisplayableImage (ipImageTest, ipImageTestDisp, hr);
		DoneTof.IN := TRUE;
	ELSIF bInitTrig AND TrigCheckTmr.Q THEN
		bError := TRUE;
		iErrorId := 402;
		fbEventlogger.bRaiseAlarm[16]:=TRUE;
		fbEventlogger.sErrorCode:= '402';
		Err.Err;
		bInitTrig := FALSE;
		TrigCheckTmr.IN := FALSE;
	END_IF
END_IF

METHOD TrigImage : BOOL
VAR_INPUT
END_VAR
fbCamera.TriggerImage();
bInitTrig := TRUE;
TrigCheckTmr.IN := TRUE;
END_METHOD

END_FUNCTION_BLOCK

// ---- POUs/FB_GlueState.TcPOU
FUNCTION_BLOCK FB_GlueState
VAR_INPUT
	stModuleHmi		: REFERENCE TO ST_ModuleHmi;
	stPlcCom		: REFERENCE TO ST_Module_PlcCom;
END_VAR
VAR
	GlueSetTmr		: TON;
	tTimeLeft		: TIME;
	sTime			: STRING;
	bDispensingSet	: BOOL;
	iDot			: INT;
END_VAR
VAR_IN_OUT
	bDetectionSucceeded : BOOL;
END_VAR

GlueSetTmr(PT := T#30M); 

tTimeLeft := GlueSetTmr.PT - GlueSetTmr.ET;
sTime := (TIME_TO_STRING(tTimeLeft));

iDot := FIND(sTime, '.');
IF iDot > 0 THEN
	stModuleHmi.sTimeSinceDispensing   := LEFT(sTime, iDot - 1);                                                  
END_IF


IF bDetectionSucceeded THEN
	stModuleHmi.bDetectionSucceeded := TRUE;
END_IF

IF tTimeLeft > T#15M AND stModuleHmi.bDetectionSucceeded AND bDispensingSet THEN
	IF NOT stModuleHmi.bProductionStageCompleted THEN
		stModuleHmi.bDispensingStageDone := TRUE;
	ELSE
		stModuleHmi.bDetectionSucceeded := FALSE;
		bDispensingSet := FALSE;
		bDetectionSucceeded := FALSE;
		stModuleHmi.bDispensingStageDone := FALSE;
		stModuleHmi.bDispensingPressed := FALSE;
	END_IF
END_IF
IF stModuleHmi.bProductionStartFailure THEN
	stModuleHmi.bDetectionSucceeded := FALSE;
	stModuleHmi.bDispensingStageDone := FALSE;
	stModuleHmi.bDispensingPressed := FALSE;
END_IF
IF stModuleHmi.bDetectionSucceeded THEN
	stModuleHmi.bAllowManDispensing := TRUE;
	bDispensingSet := TRUE;
ELSE
	stModuleHmi.bAllowManDispensing := FALSE;
END_IF

IF stModuleHmi.bDispensingPressed THEN
	GlueSetTmr.IN := TRUE;
ELSIF stModuleHmi.bDetectionSucceeded THEN
	stModuleHmi.bAllowManDispensing := TRUE;
	GlueSetTmr.IN := FALSE;
ELSE
	stModuleHmi.bAllowManDispensing := FALSE;
END_IF

IF stModuleHmi.bGlueDispensing THEN
	stPlcCom.stPlcComOut.bTriggerGluing1 := TRUE;
	stModuleHmi.bDispensingPressed := TRUE;
ELSE
	stPlcCom.stPlcComOut.bTriggerGluing1 := FALSE;
END_IF

IF stModuleHmi.bToggleDispensingPressure THEN
	stPlcCom.stPlcComOut.bGlueSelectingValve := TRUE;
ELSE
	stPlcCom.stPlcComOut.bGlueSelectingValve := FALSE;
END_IF

END_FUNCTION_BLOCK

// ---- POUs/Sts/Com/FB_DataExchangeRead.TcPOU
FUNCTION_BLOCK FB_DataExchangeRead
VAR_INPUT
	trigAdsRead		: BOOL;
	ReadData121		: REFERENCE TO ST_Vis_Laser; // // TUrhaa lukumoodissa?
	stModuleHmi		: REFERENCE TO ST_ModuleHmi;
	
	
END_VAR
VAR_OUTPUT
	stLaserPositionData		: ST_AngleData;
END_VAR
VAR
	adsWriteStatus : INT :=0; 	
	fbAdsRead		:FB_ReadAdsSymByName :=(
		sNetId :='192.168.1.10.1.1',
		nPort := 852,
		eComMode :=E_AdsComMode.eAdsComModeFastCom,
		tTimeout :=DEFAULT_ADS_TIMEOUT);
		
	bstart			: BOOL;
	delayedStart	: TON;
	resetCounter	: INT :=0;
	bAllowStart		: BOOL;
	retryDelayTON	: TON;
	bRetrytimer		: BOOL :=FALSE;
	DataLenght		: UDINT := 100;
	
	
END_VAR

//ADS Data reading case
delayedStart (IN:=TRUE, PT:=T#10S);
bAllowStart := TRUE;
IF stModuleHmi.bResetCommunication THEN
	adsWriteStatus := 30;
END_IF

CASE adsWriteStatus OF
0 : 
		IF NOT fbAdsRead.bBusy AND delayedStart.Q AND bAllowStart THEN	// Tarkastellaan toimiiko
			adsWriteStatus := 10;
		END_IF
10 :
		fbAdsRead(bRead := FALSE);
		fbAdsRead(
					sVarName := 'MAIN_VISION.stAngleData', //Luettavan tiedon osoite
					nLen := SIZEOF(stLaserPositionData), //Luettavan tiedon koko, saadaanko jostain suoraan vai pitääkö asettaa kiinteäksi. ONKO 100 JÄRKEVÄ RIITTÄVÄ TAI TOIMiva, jos sizeof ei pelaa laitetaan suoraan 100
					nDestAddr := ADR(stLaserPositionData), 	//Osoite johon kirjoitetaan luettu data
					bRead := TRUE );
		adsWriteStatus := 20;
20 :

		fbAdsRead(bRead := FALSE);
		IF NOT fbAdsRead.bBusy THEN
			IF NOT fbAdsRead.bError THEN
				adsWriteStatus := 0;
			ELSE
				adsWriteStatus := 30;
			END_IF
		END_IF
30 :
 	IF NOT bRetryTimer THEN
        retryDelayTON(IN := TRUE, PT := T#10S);
        bRetrytimer := TRUE;
    ELSE
        retryDelayTON(IN := TRUE); // keep running
    END_IF

		IF retryDelayTON.Q THEN
        	retryDelayTON(IN := FALSE); // Reset timer 
        	bRetrytimer := FALSE;

        	IF delayedStart.Q AND resetCounter < 3 AND bAllowStart THEN
            	resetCounter := resetCounter + 1;
            	adsWriteStatus := 10;         // retry write
        	ELSE
            	bAllowStart := FALSE;         // 3 attempts failed
            	adsWriteStatus := 0;          // go idle?
        END_IF
    END_IF
END_CASE

END_FUNCTION_BLOCK

// ---- POUs/HP/P_Heaters.TcPOU
PROGRAM P_Heaters
VAR
	controlSignals:			FB_ControlSignalsV2;	
	cs:						REFERENCE TO ST_CONTROL_SIGNALS_V2;

	i:	INT;
	curingStations:	ARRAY[0..4] OF FB_CuringStation;
	
	gripperOpen:	BOOL;
	gripperClosed:	BOOL;
	sliderOpen:		BOOL;
	sliderClosed:	BOOL;
	pt100Real:		REAL;

END_VAR

controlSignals(iPos := E_POS.MAIN, iMiscArea := 'Misc', ioTcHmi := HMI.cs);
cs REF= controlSignals.oControlSignals^;

curingStations[0](iStationId := 0, iDeviceId := 'Curing station 1', iControlSignals := cs.out,iGripperOpen := gripperOpen, iGripperClosed := gripperClosed, iSliderOpen := sliderOpen, iSliderClosed := sliderClosed, iPt100RawValue := pt100Real,
	ioHmi := HMI.curingStations[0], ioStaticHeaterSettings := HEATER_CONTROL_SETTINGS.settings);
	
curingStations[1](iStationId := 1, iDeviceId := 'Curing station 2', iControlSignals := cs.out,
	ioHmi := HMI.curingStations[1], ioStaticHeaterSettings := HEATER_CONTROL_SETTINGS.settings);

curingStations[2](iStationId := 2, iDeviceId := 'Curing station 3', iControlSignals := cs.out,
	ioHmi := HMI.curingStations[2], ioStaticHeaterSettings := HEATER_CONTROL_SETTINGS.settings);
	
curingStations[3](iStationId := 3, iDeviceId := 'Curing station 4', iControlSignals := cs.out,
	ioHmi := HMI.curingStations[3], ioStaticHeaterSettings := HEATER_CONTROL_SETTINGS.settings);

curingStations[4](iStationId := 4, iDeviceId := 'Curing station 5', iControlSignals := cs.out,
	ioHmi := HMI.curingStations[4], ioStaticHeaterSettings := HEATER_CONTROL_SETTINGS.settings);

END_PROGRAM

// ---- POUs/HP/CURING_STATION/FB_CuringStation.TcPOU
FUNCTION_BLOCK FB_CuringStation EXTENDS FB_StepperProgram		// This FB provides an interface for controlling the complete curing station including:
																// Slider and gripper cylinder
																// Temperature control of the heating element
																// Driving of the stepper motor and full control over the 'servo'
																// Camera + lightning
VAR_INPUT
	iGripperOpen:				BOOL;
	iGripperClosed:				BOOL;
	iSliderOpen:				BOOL;
	iSliderClosed:				BOOL;
	iRequestGripperOpen:		BOOL;
	iRequestGripperClosed:		BOOL;
	iRequestSliderOpen:			BOOL;
	iRequestSliderClosed:		BOOL;
	
	iDoStartupTest:				BOOL;
//	iStart:						BOOL;
	
	iEstopOk:					BOOL;	// 1 = System is running, no estop pressed
	iEnable:					BOOL;	// When TRUE, this sequence is possible to be run
	iStationId:					UDINT;	// Station nummer, 1..10
//	iHeatToTestTemp:			BOOL;	// When TRUE, the test program will run 
	iHeatToWorkTemp:			BOOL;	// When TRUE, will start the heating cycle
	iPt100RawValue:				REAL;	// Raw (unscaled value) of the PT100 element (or any other analog input)
	
	iDetectCoupler:				BOOL;
	iDetectMirror:				BOOL;
END_VAR
VAR_OUTPUT
	oGripperToOpen:				BOOL;
	oGripperToClosed:			BOOL;
	oSliderToOpen:				BOOL;
	oSliderToClosed:			BOOL;
	oUnderLightOn:				BOOL;
	oLaserLightOn:				BOOL;
	
	oStartupTestDone:			BOOL;
	oStartupTestFailed:			BOOL;
	oOperational:				BOOL;
	oOperationState:			E_CURING_STATION_OPERATION_STATE;
END_VAR
VAR_IN_OUT
	ioHmi:						ST_CURING_STATION_HMI;
	ioStaticHeaterSettings:		ST_CURING_STATION_HEATER_CONTROL_STATIC_SETTINGS;
END_VAR
VAR
	step:						E_CURING_STATION_SEQUENCE_STEPS;
	service:					ST_CURING_STATION_SERVICE;

	// Devices	
	cyls:						ARRAY[0..1] OF FB_Cylinder;
	heater:						FB_CuringStationHeaterControl;
	//servo:FB_Servo;

	cameraHandler:				FB_CuringStationCameraHandler;
	
	// Helper vars
	gripper:	REFERENCE TO FB_Cylinder;
	slider:		REFERENCE TO FB_Cylinder;
END_VAR
VAR PERSISTENT
	settings:					ST_CURING_STATION_SETTINGS;
END_VAR

IF (NOT IING.cycleStart) THEN
	settings := ioHmi.settings;
END_IF

service := ioHmi.service;

// Helper vars
gripper REF= cyls[0];
slider REF= cyls[1];



callMeRightBeforeSwitchCase(ADR(step));
CASE step OF
	E_CURING_STATION_SEQUENCE_STEPS.INIT:
		gotoNextStep(iDoStartupTest, E_CURING_STATION_SEQUENCE_STEPS.STARTUP_TEST_DO_ECCENTRIC_WHEEL_HOMING);

	E_CURING_STATION_SEQUENCE_STEPS.STARTUP_TEST_DO_ECCENTRIC_WHEEL_HOMING:
		gotoNextStep(TRUE, E_CURING_STATION_SEQUENCE_STEPS.STARTUP_TEST_TEST_SLIDER_TO_WORK);
	
	E_CURING_STATION_SEQUENCE_STEPS.STARTUP_TEST_TEST_SLIDER_TO_WORK:
		gotoNextStep(slider.oInOpenPos, E_CURING_STATION_SEQUENCE_STEPS.STARTUP_TEST_TEST_SLIDER_TO_HOME);

	E_CURING_STATION_SEQUENCE_STEPS.STARTUP_TEST_TEST_SLIDER_TO_HOME:
		gotoNextStep(slider.oInClosedPos, E_CURING_STATION_SEQUENCE_STEPS.STARTUP_TEST_TEST_GRIPPER_TO_WORK);
	
	E_CURING_STATION_SEQUENCE_STEPS.STARTUP_TEST_TEST_GRIPPER_TO_WORK:
		gotoNextStep(gripper.oInOpenPos, E_CURING_STATION_SEQUENCE_STEPS.STARTUP_TEST_TEST_GRIPPER_TO_HOME);

	E_CURING_STATION_SEQUENCE_STEPS.STARTUP_TEST_TEST_GRIPPER_TO_HOME:
		gotoNextStep(gripper.oInClosedPos, E_CURING_STATION_SEQUENCE_STEPS.STARTUP_TEST_TEST_UNDERLIGHT);
	
	E_CURING_STATION_SEQUENCE_STEPS.STARTUP_TEST_TEST_UNDERLIGHT:
		gotoNextStep(cameraHandler.oUnderLightTestOk, E_CURING_STATION_SEQUENCE_STEPS.STARTUP_TEST_TEST_LASER);
		gotoNextStep(cameraHandler.oUnderLightTestFailed, E_CURING_STATION_SEQUENCE_STEPS.STARTUP_TEST_FAIL);
	
	E_CURING_STATION_SEQUENCE_STEPS.STARTUP_TEST_TEST_LASER:
		gotoNextStep(cameraHandler.oLaserLightTestOk, E_CURING_STATION_SEQUENCE_STEPS.STARTUP_TEST_TEST_HEATER);
		gotoNextStep(cameraHandler.oLaserLightTestFailed, E_CURING_STATION_SEQUENCE_STEPS.STARTUP_TEST_FAIL);
	
	E_CURING_STATION_SEQUENCE_STEPS.STARTUP_TEST_TEST_HEATER:
		gotoNextStep(heater.oTestTemperatureReached, E_CURING_STATION_SEQUENCE_STEPS.STARTUP_TEST_DONE);

	E_CURING_STATION_SEQUENCE_STEPS.STARTUP_TEST_DONE:
		gotoNextStep(NOT iDoStartupTest, E_CURING_STATION_SEQUENCE_STEPS.OPERATIONAL);	

	E_CURING_STATION_SEQUENCE_STEPS.STARTUP_TEST_FAIL:
		gotoNextStep(NOT iDoStartupTest, E_CURING_STATION_SEQUENCE_STEPS.INIT);

	E_CURING_STATION_SEQUENCE_STEPS.OPERATIONAL:
		gotoNextStep(iDetectCoupler OR iDetectMirror, E_CURING_STATION_SEQUENCE_STEPS.OPERATIONAL);


ELSE
	step := E_CURING_STATION_SEQUENCE_STEPS.INIT;
END_CASE
callMeRightAfterSwitchCase(TRUE, IING.STRING_BLANK);


slider.iOpenReq := (step = E_CURING_STATION_SEQUENCE_STEPS.STARTUP_TEST_TEST_SLIDER_TO_WORK);
slider.iCloseReq := NOT slider.iOpenReq;

gripper.iOpenReq := (step = E_CURING_STATION_SEQUENCE_STEPS.STARTUP_TEST_TEST_GRIPPER_TO_WORK);
gripper.iCloseReq := NOT gripper.iOpenReq;

heater.iHeatToTestTemp := (step = E_CURING_STATION_SEQUENCE_STEPS.STARTUP_TEST_TEST_HEATER);


cameraHandler(
	iDoUnderLightTest :=		(step = E_CURING_STATION_SEQUENCE_STEPS.STARTUP_TEST_TEST_UNDERLIGHT),
	iDoLaserTest :=				(step = E_CURING_STATION_SEQUENCE_STEPS.STARTUP_TEST_TEST_LASER),
	iDetectCoupler :=			FALSE,
	iDetectMirror :=			FALSE,
	oUnderlightOn =>			oUnderlightOn,
	oLaserLightOn =>			oLaserLightOn
);



// Outputs
oStartupTestFailed := (step = E_CURING_STATION_SEQUENCE_STEPS.STARTUP_TEST_FAIL);
oStartupTestDone := (step = E_CURING_STATION_SEQUENCE_STEPS.STARTUP_TEST_DONE);
oOperational := (step = E_CURING_STATION_SEQUENCE_STEPS.OPERATIONAL);



IF (step = E_CURING_STATION_SEQUENCE_STEPS.OPERATIONAL) THEN
	oOperationState := E_CURING_STATION_OPERATION_STATE.OPERATIONAL;
ELSIF(step = E_CURING_STATION_SEQUENCE_STEPS.STARTUP_TEST_FAIL) THEN
	oOperationState := E_CURING_STATION_OPERATION_STATE.FAULTED;
END_IF

mDevices();
mHmi();

METHOD PRIVATE mDevices
{warning disable C0371}
IF (NOT __ISVALIDREF (ioHmi)) THEN
	RETURN;
END_IF

cyls[0](
	iOpenPos := iGripperOpen,
	iClosePos := iGripperClosed,
	iOpenInterLock := TRUE,
	iCloseInterlock := TRUE,
	iDeactivate := FALSE,
	iDeviceId := FC_2strConcatSeparator(iSeparator := '_', iStr1 := 'Gripper', iStr2 := iDeviceId),
	iControlSignals := iControlSignals,
	oOpen => oGripperToOpen,
	oClose => oGripperToClosed,
	ioHmi := ioHmi.cyls[0]
);


cyls[1](
	iOpenPos := iSliderOpen,
	iClosePos := iSliderClosed,
	iOpenInterLock := TRUE,
	iCloseInterlock := TRUE,
	iDeactivate := FALSE,
	iDeviceId := FC_2strConcatSeparator(iSeparator := '_', iStr1 := 'Slider', iStr2 := iDeviceId),
	iControlSignals := iControlSignals,
	oOpen => oSliderToOpen,
	oClose => oSliderToClosed,
	ioHmi := ioHmi.cyls[1]
);

heater(
	iEstopOk := iEstopOk,
	iEnable := iEnable,
//	iHeatToTestTemp :=,
	iHeatToWorkTemp := iHeatToWorkTemp,
	iPt100RawValue := iPt100RawValue,
	iControlSignals := iControlSignals,
	iDeviceId := FC_2strConcatSeparator(iSeparator := '_', iStr1 := 'Heater', iStr2 := iDeviceId),
	ioHmi := ioHmi.heater,
	ioStaticSettings := ioStaticHeaterSettings, 
);

{warning restore C0371}
END_METHOD

METHOD PRIVATE mHmi
{warning disable C0371}
IF (NOT __ISVALIDREF (ioHmi)) THEN
	RETURN;
END_IF


ioHmi.state.stationId := iStationId;
ioHmi.state.operationState := oOperationState;


ioHmi.settings := settings;
ioHmi.service := service;

{warning restore C0371}
END_METHOD

METHOD PUBLIC stepAsString : T_SHORT_STR
stepAsString := TO_STRING(step);
END_METHOD

END_FUNCTION_BLOCK

// ---- POUs/HP/CURING_STATION/HEATER/FB_CuringStationHeaterControl.TcPOU
FUNCTION_BLOCK FB_CuringStationHeaterControl EXTENDS FB_StepperProgram		// This FB is responisble for controlling the heater part of the curing station, we can be in either TEST or WORK mode
VAR_INPUT
	iEstopOk:					BOOL;	// 1 = System is running, no estop pressed
	iEnable:					BOOL;	// When TRUE, this sequence is possible to be run
	iStationId:					UDINT;	// Station nummer, 1..10
	iHeatToTestTemp:			BOOL;	// When TRUE, the test program will run 
	iHeatToWorkTemp:			BOOL;	// When TRUE, will start the heating cycle
	iPt100RawValue:				REAL;	// Raw (unscaled value) of the PT100 element (or any other analog input)
END_VAR
VAR_OUTPUT
	oTestTemperatureReached:	BOOL;	// TRUE when temperature over TEST temperature 
	oWorkTemperatureReached:	BOOL;	// TRUE when temperature over WORK temperature 
	oHeat:						BOOL;	// Heater control
	oFan:						BOOL;	// Fan control
	oTempInC:					REAL;	// Temperature in celcius
	oEnabled:					BOOL;	// When TRUe, the station is enabled
END_VAR
VAR_IN_OUT
	ioHmi:						ST_CURING_STATION_HEATER_CONTROL_HMI;
	ioStaticSettings:			ST_CURING_STATION_HEATER_CONTROL_STATIC_SETTINGS;
END_VAR
VAR
	step:						E_CURING_STATION_HEATER_CONTROL_STEPS;
	service:					ST_CURING_STATION_HEATER_CONTROL_SERVICE;
	ai:							FB_AnalogInput;
//	regularThermostat:			FB_Thermostat;
	specialThermostat:			FB_TimeProportionalThermostat;
	targetTemperature:			REAL;
	
//	staticSettings:				ST_CURING_STATION_HEATER_CONTROL_STATIC_SETTINGS;
END_VAR
VAR_STAT PERSISTENT
//	staticSettings:				ST_CURING_STATION_HEATER_CONTROL_STATIC_SETTINGS;
END_VAR

IF (NOT IING.cycleStart) THEN
	//staticSettings := ioHmi.staticSettings;
	//staticSettings:=ioStaticSettings;
	
//	staticSettings := HEATER_CONTROL_SETTINGS.settings;
END_IF

service := ioHmi.service;

callMeRightBeforeSwitchCase(ADR(step));
CASE step OF
	E_CURING_STATION_HEATER_CONTROL_STEPS.INIT:
		gotoNextStep(iCondition := iEnable AND iHeatToTestTemp, iNextStep := E_CURING_STATION_HEATER_CONTROL_STEPS.HEAT_TO_TEST_TEMP);
		gotoNextStep(iCondition := iEnable AND iHeatToWorkTemp, iNextStep := E_CURING_STATION_HEATER_CONTROL_STEPS.HEAT_TO_WORK_TEMP);
	
	E_CURING_STATION_HEATER_CONTROL_STEPS.HEAT_TO_TEST_TEMP:
		targetTemperature := ioStaticSettings.testTemperature;
		gotoNextStep(iCondition := NOT iEnable OR NOT iHeatToTestTemp, iNextStep := E_CURING_STATION_HEATER_CONTROL_STEPS.INIT);
	
	E_CURING_STATION_HEATER_CONTROL_STEPS.HEAT_TO_WORK_TEMP:
		targetTemperature := ioStaticSettings.workTemperature;
		gotoNextStep(iCondition := NOT iEnable OR NOT iHeatToWorkTemp, iNextStep := E_CURING_STATION_HEATER_CONTROL_STEPS.INIT);

	E_CURING_STATION_HEATER_CONTROL_STEPS.SAFETY_DOWN:
		gotoNextStep(iEstopOk, E_CURING_STATION_HEATER_CONTROL_STEPS.INIT);
ELSE
	step := E_CURING_STATION_HEATER_CONTROL_STEPS.INIT;
END_CASE
callMeRightAfterSwitchCase(TRUE, IING.STRING_BLANK);


// Safety check
IF (NOT iEstopOk) THEN
	gotoNextStep(iCondition := TRUE, iNextStep := E_CURING_STATION_HEATER_CONTROL_STEPS.SAFETY_DOWN);
END_IF

// Analog input
ai(iRawValue := iPt100RawValue, oScaledValue => oTempInC, iDeviceId := iDeviceId, ioHmi := ioHmi.ai);
//oTempInF := 10000;


// Temperature control/thermostat
//regularThermostat(iTargetValue := targetTemperature, iHysteresis := staticSettings.hysteresis, iMeasuredValue := ai.oScaledValue, ioHmi := ioHmi.regularThermostat);

specialThermostat(iHeat := stepInBetween(E_CURING_STATION_HEATER_CONTROL_STEPS.HEAT_TO_TEST_TEMP, E_CURING_STATION_HEATER_CONTROL_STEPS.HEAT_TO_WORK_TEMP), iTargetTemp := targetTemperature, iMeasuredTemp := ai.oScaledValue,
	iOptionalStartDelay := ULINT_TO_TIME(TIME_TO_ULINT(ioStaticSettings.cycleTime) / ioStaticSettings.nrOfStations),
	iPFactor := ioStaticSettings.pFactor, iMinPowerProcent := ioStaticSettings.minPowerProcent, iMaxPowerProcent := ioStaticSettings.maxPowerProcent, iCycleTime := ioStaticSettings.cycleTime, 
	ioHmi := iohmi.specialThermostat
);

// Controlling of actual outputs
oHeat := iEstopOk AND specialThermostat.oHeat;

// Fan follows the heating element
oFan := oHeat;


oTestTemperatureReached := FC_WithinRange(iTarget := ioStaticSettings.testTemperature, iValue := ai.oScaledValue, iRange := ioStaticSettings.hysteresis);
oWorkTemperatureReached := FC_WithinRange(iTarget := ioStaticSettings.workTemperature, iValue := ai.oScaledValue, iRange := ioStaticSettings.hysteresis);

oEnabled := iEnable;

mStatistics();

mHmi();

METHOD PRIVATE mHmi
{warning disable C0371}
IF (NOT __ISVALIDREF (ioHmi)) THEN
	RETURN;
END_IF

//ioHmi.staticSettings := staticSettings;
ioHmi.service := service;

ioHmi.state.enabled := oEnabled;
ioHmi.state.heat := oHeat;
ioHmi.state.fan := oFan;
ioHmi.state.tempInC := oTempInC;
//ioHmi.state.tempInF := oTempInF;


ioHmi.state.testTemperatureReached := oTestTemperatureReached;
ioHmi.state.workTemperatureReached := oWorkTemperatureReached;

ioHmi.state.stationId := iStationId;


{warning restore C0371}
END_METHOD

METHOD mStatistics : BOOL
VAR_INST
	switchHeatOnCount:		FB_EventCounter;
	heatDurationOnCount:	FB_DurationCounter;
END_VAR
switchHeatOnCount(iEvent := oHeat);

heatDurationOnCount(iSignal := oHeat);
END_METHOD

METHOD PUBLIC stepAsString : T_SHORT_STR
stepAsString := TO_STRING(step);
END_METHOD

END_FUNCTION_BLOCK

// ---- POUs/HP/CURING_STATION/VISION/FB_CuringStationCameraHandler.TcPOU
FUNCTION_BLOCK FB_CuringStationCameraHandler EXTENDS FB_StepperProgram	
VAR_INPUT
	iDoUnderLightTest:		BOOL;
	iDoLaserTest:			BOOL;
	iDetectCoupler:			BOOL;
	iDetectMirror:			BOOL;
	
	iCouplerProcessor:		I_ImageProcessor;		// FB implementing
	iMirrorProcessor:		I_MirrorImageProcessor;
	
END_VAR
VAR_OUTPUT
	oUnderLightTestOk:			BOOL;
	oUnderLightTestFailed:		BOOL;
	oLaserLightTestOk:			BOOL;
	oLaserLightTestFailed:		BOOL;

	oCouplerDetectDone:			BOOL;
	oCouplerDetectFailed:		BOOL;

	oHmi:						ST_NORMAL_CAM_HANDLER_HMI;
	
	oUnderlightOn:				BOOL;
	oLaserLightOn:				BOOL;
END_VAR
VAR_IN_OUT
END_VAR
VAR
	step:					E_NORMAL_CAM_HANDLER_SEQ_STEPS;
	service:				ST_NORMAL_CAM_HANDLER_SERVICE;
	
	visionState:			ETcVnCameraState;
	gigECameraHandler:		FB_GigECamHandler;
	hResult:				HRESULT;
	
	rectangleArea:			TcVnRectangle_UDINT;
	rawImageCopy:			ITcVnImage;				// Image of either under light/laser
	processedImage:			ITcVnImage;
	displayableProcessedImage:	ITcVnDisplayableImage;

	averagePixelValue:		TcVnVector4_LREAL;
	
	reset:					BOOL;
END_VAR
VAR PERSISTENT
	settings:				ST_NORMAL_CAM_HANDLER_SETTINGS;
END_VAR

reset := iControlSignals.resetPulse;



callMeRightBeforeSwitchCase(ADR(step));
CASE step OF
	E_NORMAL_CAM_HANDLER_SEQ_STEPS.INIT:
		gotoNextStep(iDoUnderLightTest OR service.doUnderLightTest, E_NORMAL_CAM_HANDLER_SEQ_STEPS.UNDER_LIGHT_TEST_ENABLE_LIGHT);
		gotoNextStep(iDoLaserTest OR service.doLaserTest, E_NORMAL_CAM_HANDLER_SEQ_STEPS.LASER_LIGHT_TEST_ENABLE_LIGHT);
		gotoNextStep(iDetectCoupler, E_NORMAL_CAM_HANDLER_SEQ_STEPS.COUPLER_DETECT_ENABLE_LIGHT);
		gotoNextStep(iDetectMirror, E_NORMAL_CAM_HANDLER_SEQ_STEPS.MIRROR_DETECT_ENABLE_LIGHT);


// --------------------------------- UNDER LIGHT TEST	
	E_NORMAL_CAM_HANDLER_SEQ_STEPS.UNDER_LIGHT_TEST_ENABLE_LIGHT:
		gotoNextStep(isTimeExpired(T#500MS), E_NORMAL_CAM_HANDLER_SEQ_STEPS.UNDER_LIGHT_TEST_IMAGE_ACQUIRE);
	
	E_NORMAL_CAM_HANDLER_SEQ_STEPS.UNDER_LIGHT_TEST_IMAGE_ACQUIRE:
		gotoNextStep(gigECameraHandler.oImageAcquired, E_NORMAL_CAM_HANDLER_SEQ_STEPS.UNDER_LIGHT_TEST_IMAGE_PROCESSING);
		gotoNextStep(gigECameraHandler.oError, E_NORMAL_CAM_HANDLER_SEQ_STEPS.UNDER_LIGHT_TEST_FAILED);
	
	E_NORMAL_CAM_HANDLER_SEQ_STEPS.UNDER_LIGHT_TEST_IMAGE_PROCESSING:
		hResult := F_VN_CopyImage(gigECameraHandler.oRawImage, rawImageCopy, hrPrev := hResult);
		rectangleArea.nHeight := settings.underLightTest.height;
		rectangleArea.nWidth := settings.underLightTest.width;
		rectangleArea.nX := settings.underLightTest.x;
		rectangleArea.nY := settings.underLightTest.y;
		
		hResult := F_VN_SetRoi_TcVnRectangle_UDINT(stRoi := rectangleArea, ipDestImage := rawImageCopy, hrPrev := hResult);
		hResult := F_VN_ImageAverage(ipSrcImage := rawImageCopy, aAverage := averagePixelValue, hrPrev := hResult);
		hResult := F_VN_ResetRoi(ipImage := rawImageCopy, hrPrev := hResult);
		
		gotoNextStep((averagePixelValue[0] >= settings.underLightTest.threshold), E_NORMAL_CAM_HANDLER_SEQ_STEPS.UNDER_LIGHT_TEST_OK);  			
		gotoNextStep((averagePixelValue[0] < settings.underLightTest.threshold), E_NORMAL_CAM_HANDLER_SEQ_STEPS.UNDER_LIGHT_TEST_FAILED);
	
	E_NORMAL_CAM_HANDLER_SEQ_STEPS.UNDER_LIGHT_TEST_OK:
		gotoNextStep(NOT iDoUnderLightTest, E_NORMAL_CAM_HANDLER_SEQ_STEPS.INIT);

	E_NORMAL_CAM_HANDLER_SEQ_STEPS.UNDER_LIGHT_TEST_FAILED:
		gotoNextStep(NOT iDoUnderLightTest, E_NORMAL_CAM_HANDLER_SEQ_STEPS.INIT);
		
		
// --------------------------------- LASER LIGHT TEST
	E_NORMAL_CAM_HANDLER_SEQ_STEPS.LASER_LIGHT_TEST_ENABLE_LIGHT:
		gotoNextStep(isTimeExpired(T#250MS), E_NORMAL_CAM_HANDLER_SEQ_STEPS.LASER_LIGHT_TEST_IMAGE_ACQUIRE);

	E_NORMAL_CAM_HANDLER_SEQ_STEPS.LASER_LIGHT_TEST_IMAGE_ACQUIRE:
		gotoNextStep(gigECameraHandler.oImageAcquired, E_NORMAL_CAM_HANDLER_SEQ_STEPS.LASER_LIGHT_TEST_IMAGE_PROCESSING);
		gotoNextStep(gigECameraHandler.oError, E_NORMAL_CAM_HANDLER_SEQ_STEPS.LASER_LIGHT_TEST_FAILED);
	
	E_NORMAL_CAM_HANDLER_SEQ_STEPS.LASER_LIGHT_TEST_IMAGE_PROCESSING:
		hResult := F_VN_CopyImage(gigECameraHandler.oRawImage, rawImageCopy, hrPrev := hResult);
		rectangleArea.nHeight := settings.laserTest.height;
		rectangleArea.nWidth := settings.laserTest.width;
		rectangleArea.nX := settings.laserTest.x;
		rectangleArea.nY := settings.laserTest.y;
		
		hResult := F_VN_SetRoi_TcVnRectangle_UDINT(stRoi := rectangleArea, ipDestImage := rawImageCopy, hrPrev := hResult);
		hResult := F_VN_ImageAverage(ipSrcImage := rawImageCopy, aAverage := averagePixelValue, hrPrev := hResult);
		hResult := F_VN_ResetRoi(ipImage := rawImageCopy, hrPrev := hResult);
		gotoNextStep((averagePixelValue[0] >= settings.laserTest.threshold), E_NORMAL_CAM_HANDLER_SEQ_STEPS.LASER_LIGHT_TEST_OK);  			
		gotoNextStep((averagePixelValue[0] < settings.laserTest.threshold), E_NORMAL_CAM_HANDLER_SEQ_STEPS.LASER_LIGHT_TEST_FAILED);
	
	E_NORMAL_CAM_HANDLER_SEQ_STEPS.LASER_LIGHT_TEST_OK:
		gotoNextStep(NOT iDoUnderLightTest, E_NORMAL_CAM_HANDLER_SEQ_STEPS.INIT);

	E_NORMAL_CAM_HANDLER_SEQ_STEPS.LASER_LIGHT_TEST_FAILED:
		gotoNextStep(NOT iDoUnderLightTest, E_NORMAL_CAM_HANDLER_SEQ_STEPS.INIT);


// --------------------------------- COUPLER DETECT
	E_NORMAL_CAM_HANDLER_SEQ_STEPS.COUPLER_DETECT_ENABLE_LIGHT:
		gotoNextStep(isTimeExpired(T#500MS), E_NORMAL_CAM_HANDLER_SEQ_STEPS.COUPLER_DETECT_IMAGE_ACQUIRE);

